//Place your alarm trigger logic here. 
IF io_mapping.cct_3342_b.scaled_value < opc.popa_0082_cct_3342_b_low_setpoint THEN
    cct_3342_b_low.trigger := TRUE;
    ELSE
        cct_3342_b_low.trigger := FALSE;
END_IF
	
//cct_3342-----------------------------------------------------------------------------------------------------
//Instantiate the alarm block, and map the inputs from the OPC GVL
cct_3342_b_high();
cct_3342_b_high.alm_ack:=opc.popa_0082_alarm_ack;
cct_3342_b_high.reset:=opc.popa_0082_alarm_reset;
cct_3342_b_high.priority:=opc.popa_0082_cct_3342_b_high_priority;
cct_3342_b_high.delay_setpoint:=opc.popa_0082_cct_3342_b_high_setpoint;
cct_3342_b_high.enable:=opc.popa_0082_cct_3342_b_high_enable;

//Timer delay elapsed
cct_3342_b_high.delay_ton_et;

//Place your alarm trigger logic here. 
IF io_mapping.cct_3342_b.scaled_value > opc.popa_0082_cct_3342_b_high_setpoint THEN
    cct_3342_b_high.trigger := TRUE;
    ELSE
        cct_3342_b_high.trigger := FALSE;
END_IF
	
//cct_3342-----------------------------------------------------------------------------------------------------
//Instantiate the alarm block, and map the inputs from the OPC GVL
cct_3342_b_high_high();
cct_3342_b_high_high.alm_ack:=opc.popa_0082_alarm_ack;
cct_3342_b_high_high.reset:=opc.popa_0082_alarm_reset;
cct_3342_b_high_high.priority:=opc.popa_0082_cct_3342_b_high_high_priority;
cct_3342_b_high_high.delay_setpoint:=opc.popa_0082_cct_3342_b_high_high_setpoint;
cct_3342_b_high_high.enable:=opc.popa_0082_cct_3342_b_high_high_enable;

//Timer delay elapsed
cct_3342_b_high_high.delay_ton_et;

//Place your alarm trigger logic here. 
IF io_mapping.cct_3342_b.scaled_value >= opc.popa_0082_cct_3342_b_high_high_setpoint THEN
    cct_3342_b_high_high.trigger := TRUE;
    ELSE
        cct_3342_b_high_high.trigger := FALSE;
END_IF

(*
//cct_3413-----------------------------------------------------------------------------------------------------
//Instantiate the alarm block, and map the inputs from the OPC GVL
cct_3413_b_low_low();
cct_3413_b_low_low.alm_ack:=opc.popa_0082_alarm_ack;
cct_3413_b_low_low.reset:=opc.popa_0082_alarm_reset;
cct_3413_b_low_low.priority:=opc.popa_0092_cct_3413_b_low_low_priority;
cct_3413_b_low_low.delay_setpoint:=opc.popa_0092_cct_3413_b_low_low_setpoint;
cct_3413_b_low_low.enable:=opc.popa_0092_cct_3413_b_low_low_enable;

//Timer delay elapsed
cct_3413_b_low_low.delay_ton_et;

//Place your alarm trigger logic here. 
IF io_mapping.cct_3413_b.scaled_value <= opc.popa_0092_cct_3413_b_low_low_setpoint THEN
    cct_3413_b_low_low.trigger := TRUE;
    ELSE
        cct_3413_b_low_low.trigger := FALSE;
END_IF
	
//cct_3413-----------------------------------------------------------------------------------------------------
//Instantiate the alarm block, and map the inputs from the OPC GVL
cct_3413_b_low();
cct_3413_b_low.alm_ack:=opc.popa_0082_alarm_ack;
cct_3413_b_low.reset:=opc.popa_0082_alarm_reset;
cct_3413_b_low.priority:=opc.popa_0092_cct_3413_b_low_priority;
cct_3413_b_low.delay_setpoint:=opc.popa_0092_cct_3413_b_low_setpoint;
cct_3413_b_low.enable:=opc.popa_0092_cct_3413_b_low_enable;

//Timer delay elapsed
cct_3413_b_low.delay_ton_et;

//Place your alarm trigger logic here. 
IF io_mapping.cct_3413_b.scaled_value < opc.popa_0092_cct_3413_b_low_setpoint THEN
    cct_3413_b_low.trigger := TRUE;
    ELSE
        cct_3413_b_low.trigger := FALSE;
END_IF
	
//cct_3413-----------------------------------------------------------------------------------------------------
//Instantiate the alarm block, and map the inputs from the OPC GVL
cct_3413_b_high();
cct_3413_b_high.alm_ack:=opc.popa_0082_alarm_ack;
cct_3413_b_high.reset:=opc.popa_0082_alarm_reset;
cct_3413_b_high.priority:=opc.popa_0092_cct_3413_b_high_priority;
cct_3413_b_high.delay_setpoint:=opc.popa_0092_cct_3413_b_high_setpoint;
cct_3413_b_high.enable:=opc.popa_0092_cct_3413_b_high_enable;

//Timer delay elapsed
cct_3413_b_high.delay_ton_et;

//Place your alarm trigger logic here. 
IF io_mapping.cct_3413_b.scaled_value > opc.popa_0092_cct_3413_b_high_setpoint THEN
    cct_3413_b_high.trigger := TRUE;
    ELSE
        cct_3413_b_high.trigger := FALSE;
END_IF
	
//cct_3413-----------------------------------------------------------------------------------------------------
//Instantiate the alarm block, and map the inputs from the OPC GVL
cct_3413_b_high_high();
cct_3413_b_high_high.alm_ack:=opc.popa_0082_alarm_ack;
cct_3413_b_high_high.reset:=opc.popa_0082_alarm_reset;
cct_3413_b_high_high.priority:=opc.popa_0092_cct_3413_b_high_high_priority;
cct_3413_b_high_high.delay_setpoint:=opc.popa_0092_cct_3413_b_high_high_setpoint;
cct_3413_b_high_high.enable:=opc.popa_0092_cct_3413_b_high_high_enable;

//Timer delay elapsed
cct_3413_b_high_high.delay_ton_et;

//Place your alarm trigger logic here. 
IF io_mapping.cct_3413_b.scaled_value >= opc.popa_0092_cct_3413_b_high_high_setpoint THEN
    cct_3413_b_high_high.trigger := TRUE;
    ELSE
        cct_3413_b_high_high.trigger := FALSE;
END_IF

*)

//ft_3122-----------------------------------------------------------------------------------------------------
//Instantiate the alarm block, and map the inputs from the OPC GVL
ft_3122_b_low_low();
ft_3122_b_low_low.alm_ack:=opc.popa_0082_alarm_ack;
ft_3122_b_low_low.reset:=opc.popa_0082_alarm_reset;
ft_3122_b_low_low.priority:=opc.popa_0082_ft_3122_b_low_low_priority;
ft_3122_b_low_low.delay_setpoint:=opc.popa_0082_ft_3122_b_low_low_setpoint;
ft_3122_b_low_low.enable:=opc.popa_0082_ft_3122_b_low_low_enable;

//Timer delay elapsed
ft_3122_b_low_low.delay_ton_et;

//Place your alarm trigger logic here. 
IF io_mapping.ft_3122_b.scaled_value <= opc.popa_0082_ft_3122_b_low_low_setpoint THEN
    ft_3122_b_low_low.trigger := TRUE;
    ELSE
        ft_3122_b_low_low.trigger := FALSE;
END_IF
	
//ft_3122-----------------------------------------------------------------------------------------------------
//Instantiate the alarm block, and map the inputs from the OPC GVL
ft_3122_b_low();
ft_3122_b_low.alm_ack:=opc.popa_0082_alarm_ack;
ft_3122_b_low.reset:=opc.popa_0082_alarm_reset;
ft_3122_b_low.priority:=opc.popa_0082_ft_3122_b_low_priority;
ft_3122_b_low.delay_setpoint:=opc.popa_0082_ft_3122_b_low_setpoint;
ft_3122_b_low.enable:=opc.popa_0082_ft_3122_b_low_enable;

//Timer delay elapsed
ft_3122_b_low.delay_ton_et;

//Place your alarm trigger logic here. 
IF io_mapping.ft_3122_b.scaled_value < opc.popa_0082_ft_3122_b_low_setpoint THEN
    ft_3122_b_low.trigger := TRUE;
    ELSE
        ft_3122_b_low.trigger := FALSE;
END_IF
	
//ft_3122-----------------------------------------------------------------------------------------------------
//Instantiate the alarm block, and map the inputs from the OPC GVL
ft_3122_b_high();
ft_3122_b_high.alm_ack:=opc.popa_0082_alarm_ack;
ft_3122_b_high.reset:=opc.popa_0082_alarm_reset;
ft_3122_b_high.priority:=opc.popa_0082_ft_3122_b_high_priority;
ft_3122_b_high.delay_setpoint:=opc.popa_0082_ft_3122_b_high_setpoint;
ft_3122_b_high.enable:=opc.popa_0082_ft_3122_b_high_enable;

//Timer delay elapsed
ft_3122_b_high.delay_ton_et;

//Place your alarm trigger logic here. 
IF io_mapping.ft_3122_b.scaled_value > opc.popa_0082_ft_3122_b_high_setpoint THEN
    ft_3122_b_high.trigger := TRUE;
    ELSE
        ft_3122_b_high.trigger := FALSE;
END_IF
	
//ft_3122-----------------------------------------------------------------------------------------------------
//Instantiate the alarm block, and map the inputs from the OPC GVL
ft_3122_b_high_high();
ft_3122_b_high_high.alm_ack:=opc.popa_0082_alarm_ack;
ft_3122_b_high_high.reset:=opc.popa_0082_alarm_reset;
ft_3122_b_high_high.priority:=opc.popa_0082_ft_3122_b_high_high_priority;
ft_3122_b_high_high.delay_setpoint:=opc.popa_0082_ft_3122_b_high_high_setpoint;
ft_3122_b_high_high.enable:=opc.popa_0082_ft_3122_b_high_high_enable;

//Timer delay elapsed
ft_3122_b_high_high.delay_ton_et;

//Place your alarm trigger logic here. 
IF io_mapping.ft_3122_b.scaled_value >= opc.popa_0082_ft_3122_b_high_high_setpoint THEN
    ft_3122_b_high_high.trigger := TRUE;
    ELSE
        ft_3122_b_high_high.trigger := FALSE;
END_IF


//ft_3222-----------------------------------------------------------------------------------------------------
//Instantiate the alarm block, and map the inputs from the OPC GVL
ft_3222_b_low_low();
ft_3222_b_low_low.alm_ack:=opc.popa_0082_alarm_ack;
ft_3222_b_low_low.reset:=opc.popa_0082_alarm_reset;
ft_3222_b_low_low.priority:=opc.popa_0082_ft_3222_b_low_low_priority;
ft_3222_b_low_low.delay_setpoint:=opc.popa_0082_ft_3222_b_low_low_setpoint;
ft_3222_b_low_low.enable:=opc.popa_0082_ft_3222_b_low_low_enable;

//Timer delay elapsed
ft_3222_b_low_low.delay_ton_et;

//Place your alarm trigger logic here. 
IF io_mapping.ft_3222_b.scaled_value <= opc.popa_0082_ft_3222_b_low_low_setpoint THEN
    ft_3222_b_low_low.trigger := TRUE;
    ELSE
        ft_3222_b_low_low.trigger := FALSE;
END_IF
	
//ft_3222-----------------------------------------------------------------------------------------------------
//Instantiate the alarm block, and map the inputs from the OPC GVL
ft_3222_b_low();
ft_3222_b_low.alm_ack:=opc.popa_0082_alarm_ack;
ft_3222_b_low.reset:=opc.popa_0082_alarm_reset;
ft_3222_b_low.priority:=opc.popa_0082_ft_3222_b_low_priority;
ft_3222_b_low.delay_setpoint:=opc.popa_0082_ft_3222_b_low_setpoint;
ft_3222_b_low.enable:=opc.popa_0082_ft_3222_b_low_enable;

//Timer delay elapsed
ft_3222_b_low.delay_ton_et;

//Place your alarm trigger logic here. 
IF io_mapping.ft_3222_b.scaled_value < opc.popa_0082_ft_3222_b_low_setpoint THEN
    ft_3222_b_low.trigger := TRUE;
    ELSE
        ft_3222_b_low.trigger := FALSE;
END_IF
	
//ft_3222-----------------------------------------------------------------------------------------------------
//Instantiate the alarm block, and map the inputs from the OPC GVL
ft_3222_b_high();
ft_3222_b_high.alm_ack:=opc.popa_0082_alarm_ack;
ft_3222_b_high.reset:=opc.popa_0082_alarm_reset;
ft_3222_b_high.priority:=opc.popa_0082_ft_3222_b_high_priority;
ft_3222_b_high.delay_setpoint:=opc.popa_0082_ft_3222_b_high_setpoint;
ft_3222_b_high.enable:=opc.popa_0082_ft_3222_b_high_enable;

//Timer delay elapsed
ft_3222_b_high.delay_ton_et;

//Place your alarm trigger logic here. 
IF io_mapping.ft_3222_b.scaled_value > opc.popa_0082_ft_3222_b_high_setpoint THEN
    ft_3222_b_high.trigger := TRUE;
    ELSE
        ft_3222_b_high.trigger := FALSE;
END_IF
	
//ft_3222-----------------------------------------------------------------------------------------------------
//Instantiate the alarm block, and map the inputs from the OPC GVL
ft_3222_b_high_high();
ft_3222_b_high_high.alm_ack:=opc.popa_0082_alarm_ack;
ft_3222_b_high_high.reset:=opc.popa_0082_alarm_reset;
ft_3222_b_high_high.priority:=opc.popa_0082_ft_3222_b_high_high_priority;
ft_3222_b_high_high.delay_setpoint:=opc.popa_0082_ft_3222_b_high_high_setpoint;
ft_3222_b_high_high.enable:=opc.popa_0082_ft_3222_b_high_high_enable;

//Timer delay elapsed
ft_3222_b_high_high.delay_ton_et;

//Place your alarm trigger logic here. 
IF io_mapping.ft_3222_b.scaled_value >= opc.popa_0082_ft_3222_b_high_high_setpoint THEN
    ft_3222_b_high_high.trigger := TRUE;
    ELSE
        ft_3222_b_high_high.trigger := FALSE;
END_IF


//ft_3322-----------------------------------------------------------------------------------------------------
//Instantiate the alarm block, and map the inputs from the OPC GVL
ft_3322_b_low_low();
ft_3322_b_low_low.alm_ack:=opc.popa_0082_alarm_ack;
ft_3322_b_low_low.reset:=opc.popa_0082_alarm_reset;
ft_3322_b_low_low.priority:=opc.popa_0082_ft_3322_b_low_low_priority;
ft_3322_b_low_low.delay_setpoint:=opc.popa_0082_ft_3322_b_low_low_setpoint;
ft_3322_b_low_low.enable:=opc.popa_0082_ft_3322_b_low_low_enable;

//Timer delay elapsed
ft_3322_b_low_low.delay_ton_et;

//Place your alarm trigger logic here. 
IF io_mapping.ft_3322_b.scaled_value <= opc.popa_0082_ft_3322_b_low_low_setpoint THEN
    ft_3322_b_low_low.trigger := TRUE;
    ELSE
        ft_3322_b_low_low.trigger := FALSE;
END_IF
	
//ft_3322-----------------------------------------------------------------------------------------------------
//Instantiate the alarm block, and map the inputs from the OPC GVL
ft_3322_b_low();
ft_3322_b_low.alm_ack:=opc.popa_0082_alarm_ack;
ft_3322_b_low.reset:=opc.popa_0082_alarm_reset;
ft_3322_b_low.priority:=opc.popa_0082_ft_3322_b_low_priority;
ft_3322_b_low.delay_setpoint:=opc.popa_0082_ft_3322_b_low_setpoint;
ft_3322_b_low.enable:=opc.popa_0082_ft_3322_b_low_enable;

//Timer delay elapsed
ft_3322_b_low.delay_ton_et;

//Place your alarm trigger logic here. 
IF io_mapping.ft_3322_b.scaled_value < opc.popa_0082_ft_3322_b_low_setpoint THEN
    ft_3322_b_low.trigger := TRUE;
    ELSE
        ft_3322_b_low.trigger := FALSE;
END_IF
	
//ft_3322-----------------------------------------------------------------------------------------------------
//Instantiate the alarm block, and map the inputs from the OPC GVL
ft_3322_b_high();
ft_3322_b_high.alm_ack:=opc.popa_0082_alarm_ack;
ft_3322_b_high.reset:=opc.popa_0082_alarm_reset;
ft_3322_b_high.priority:=opc.popa_0082_ft_3322_b_high_priority;
ft_3322_b_high.delay_setpoint:=opc.popa_0082_ft_3322_b_high_setpoint;
ft_3322_b_high.enable:=opc.popa_0082_ft_3322_b_high_enable;

//Timer delay elapsed
ft_3322_b_high.delay_ton_et;

//Place your alarm trigger logic here. 
IF io_mapping.ft_3322_b.scaled_value > opc.popa_0082_ft_3322_b_high_setpoint THEN
    ft_3322_b_high.trigger := TRUE;
    ELSE
        ft_3322_b_high.trigger := FALSE;
END_IF
	
//ft_3322-----------------------------------------------------------------------------------------------------
//Instantiate the alarm block, and map the inputs from the OPC GVL
ft_3322_b_high_high();
ft_3322_b_high_high.alm_ack:=opc.popa_0082_alarm_ack;
ft_3322_b_high_high.reset:=opc.popa_0082_alarm_reset;
ft_3322_b_high_high.priority:=opc.popa_0082_ft_3322_b_high_high_priority;
ft_3322_b_high_high.delay_setpoint:=opc.popa_0082_ft_3322_b_high_high_setpoint;
ft_3322_b_high_high.enable:=opc.popa_0082_ft_3322_b_high_high_enable;

//Timer delay elapsed
ft_3322_b_high_high.delay_ton_et;

//Place your alarm trigger logic here. 
IF io_mapping.ft_3322_b.scaled_value >= opc.popa_0082_ft_3322_b_high_high_setpoint THEN
    ft_3322_b_high_high.trigger := TRUE;
    ELSE
        ft_3322_b_high_high.trigger := FALSE;
END_IF


//lt_3102-----------------------------------------------------------------------------------------------------
//Instantiate the alarm block, and map the inputs from the OPC GVL
lt_3102_b_low_low();
lt_3102_b_low_low.alm_ack:=opc.popa_0082_alarm_ack;
lt_3102_b_low_low.reset:=opc.popa_0082_alarm_reset;
lt_3102_b_low_low.priority:=opc.popa_0082_lt_3102_b_low_low_priority;
lt_3102_b_low_low.delay_setpoint:=opc.popa_0082_lt_3102_b_low_low_setpoint;
lt_3102_b_low_low.enable:=opc.popa_0082_lt_3102_b_low_low_enable;

//Timer delay elapsed
lt_3102_b_low_low.delay_ton_et;

//Place your alarm trigger logic here. 
IF io_mapping.lt_3102_b.scaled_value <= opc.popa_0082_lt_3102_b_low_low_setpoint THEN
    lt_3102_b_low_low.trigger := TRUE;
    ELSE
        lt_3102_b_low_low.trigger := FALSE;
END_IF
	
//lt_3102-----------------------------------------------------------------------------------------------------
//Instantiate the alarm block, and map the inputs from the OPC GVL
lt_3102_b_low();
lt_3102_b_low.alm_ack:=opc.popa_0082_alarm_ack;
lt_3102_b_low.reset:=opc.popa_0082_alarm_reset;
lt_3102_b_low.priority:=opc.popa_0082_lt_3102_b_low_priority;
lt_3102_b_low.delay_setpoint:=opc.popa_0082_lt_3102_b_low_setpoint;
lt_3102_b_low.enable:=opc.popa_0082_lt_3102_b_low_enable;

//Timer delay elapsed
lt_3102_b_low.delay_ton_et;

//Place your alarm trigger logic here. 
IF io_mapping.lt_3102_b.scaled_value < opc.popa_0082_lt_3102_b_low_setpoint THEN
    lt_3102_b_low.trigger := TRUE;
    ELSE
        lt_3102_b_low.trigger := FALSE;
END_IF
	
//lt_3102-----------------------------------------------------------------------------------------------------
//Instantiate the alarm block, and map the inputs from the OPC GVL
lt_3102_b_high();
lt_3102_b_high.alm_ack:=opc.popa_0082_alarm_ack;
lt_3102_b_high.reset:=opc.popa_0082_alarm_reset;
lt_3102_b_high.priority:=opc.popa_0082_lt_3102_b_high_priority;
lt_3102_b_high.delay_setpoint:=opc.popa_0082_lt_3102_b_high_setpoint;
lt_3102_b_high.enable:=opc.popa_0082_lt_3102_b_high_enable;

//Timer delay elapsed
lt_3102_b_high.delay_ton_et;

//Place your alarm trigger logic here. 
IF io_mapping.lt_3102_b.scaled_value > opc.popa_0082_lt_3102_b_high_setpoint THEN
    lt_3102_b_high.trigger := TRUE;
    ELSE
        lt_3102_b_high.trigger := FALSE;
END_IF
	
//lt_3102-----------------------------------------------------------------------------------------------------
//Instantiate the alarm block, and map the inputs from the OPC GVL
lt_3102_b_high_high();
lt_3102_b_high_high.alm_ack:=opc.popa_0082_alarm_ack;
lt_3102_b_high_high.reset:=opc.popa_0082_alarm_reset;
lt_3102_b_high_high.priority:=opc.popa_0082_lt_3102_b_high_high_priority;
lt_3102_b_high_high.delay_setpoint:=opc.popa_0082_lt_3102_b_high_high_setpoint;
lt_3102_b_high_high.enable:=opc.popa_0082_lt_3102_b_high_high_enable;

//Timer delay elapsed
lt_3102_b_high_high.delay_ton_et;

//Place your alarm trigger logic here. 
IF io_mapping.lt_3102_b.scaled_value >= opc.popa_0082_lt_3102_b_high_high_setpoint THEN
    lt_3102_b_high_high.trigger := TRUE;
    ELSE
        lt_3102_b_high_high.trigger := FALSE;
END_IF


//lt_3202-----------------------------------------------------------------------------------------------------
//Instantiate the alarm block, and map the inputs from the OPC GVL
lt_3202_b_low_low();
lt_3202_b_low_low.alm_ack:=opc.popa_0082_alarm_ack;
lt_3202_b_low_low.reset:=opc.popa_0082_alarm_reset;
lt_3202_b_low_low.priority:=opc.popa_0082_lt_3202_b_low_low_priority;
lt_3202_b_low_low.delay_setpoint:=opc.popa_0082_lt_3202_b_low_low_setpoint;
lt_3202_b_low_low.enable:=opc.popa_0082_lt_3202_b_low_low_enable;

//Timer delay elapsed
lt_3202_b_low_low.delay_ton_et;

//Place your alarm trigger logic here. 
IF io_mapping.lt_3202_b.scaled_value <= opc.popa_0082_lt_3202_b_low_low_setpoint THEN
    lt_3202_b_low_low.trigger := TRUE;
    ELSE
        lt_3202_b_low_low.trigger := FALSE;
END_IF
	
//lt_3202-----------------------------------------------------------------------------------------------------
//Instantiate the alarm block, and map the inputs from the OPC GVL
lt_3202_b_low();
lt_3202_b_low.alm_ack:=opc.popa_0082_alarm_ack;
lt_3202_b_low.reset:=opc.popa_0082_alarm_reset;
lt_3202_b_low.priority:=opc.popa_0082_lt_3202_b_low_priority;
lt_3202_b_low.delay_setpoint:=opc.popa_0082_lt_3202_b_low_setpoint;
lt_3202_b_low.enable:=opc.popa_0082_lt_3202_b_low_enable;

//Timer delay elapsed
lt_3202_b_low.delay_ton_et;

//Place your alarm trigger logic here. 
IF io_mapping.lt_3202_b.scaled_value < opc.popa_0082_lt_3202_b_low_setpoint THEN
    lt_3202_b_low.trigger := TRUE;
    ELSE
        lt_3202_b_low.trigger := FALSE;
END_IF
	
//lt_3202-----------------------------------------------------------------------------------------------------
//Instantiate the alarm block, and map the inputs from the OPC GVL
lt_3202_b_high();
lt_3202_b_high.alm_ack:=opc.popa_0082_alarm_ack;
lt_3202_b_high.reset:=opc.popa_0082_alarm_reset;
lt_3202_b_high.priority:=opc.popa_0082_lt_3202_b_high_priority;
lt_3202_b_high.delay_setpoint:=opc.popa_0082_lt_3202_b_high_setpoint;
lt_3202_b_high.enable:=opc.popa_0082_lt_3202_b_high_enable;

//Timer delay elapsed
lt_3202_b_high.delay_ton_et;

//Place your alarm trigger logic here. 
IF io_mapping.lt_3202_b.scaled_value > opc.popa_0082_lt_3202_b_high_setpoint THEN
    lt_3202_b_high.trigger := TRUE;
    ELSE
        lt_3202_b_high.trigger := FALSE;
END_IF
	
//lt_3202-----------------------------------------------------------------------------------------------------
//Instantiate the alarm block, and map the inputs from the OPC GVL
lt_3202_b_high_high();
lt_3202_b_high_high.alm_ack:=opc.popa_0082_alarm_ack;
lt_3202_b_high_high.reset:=opc.popa_0082_alarm_reset;
lt_3202_b_high_high.priority:=opc.popa_0082_lt_3202_b_high_high_priority;
lt_3202_b_high_high.delay_setpoint:=opc.popa_0082_lt_3202_b_high_high_setpoint;
lt_3202_b_high_high.enable:=opc.popa_0082_lt_3202_b_high_high_enable;

//Timer delay elapsed
lt_3202_b_high_high.delay_ton_et;

//Place your alarm trigger logic here. 
IF io_mapping.lt_3202_b.scaled_value >= opc.popa_0082_lt_3202_b_high_high_setpoint THEN
    lt_3202_b_high_high.trigger := TRUE;
    ELSE
        lt_3202_b_high_high.trigger := FALSE;
END_IF


//lt_3302-----------------------------------------------------------------------------------------------------
//Instantiate the alarm block, and map the inputs from the OPC GVL
lt_3302_b_low_low();
lt_3302_b_low_low.alm_ack:=opc.popa_0082_alarm_ack;
lt_3302_b_low_low.reset:=opc.popa_0082_alarm_reset;
lt_3302_b_low_low.priority:=opc.popa_0082_lt_3302_b_low_low_priority;
lt_3302_b_low_low.delay_setpoint:=opc.popa_0082_lt_3302_b_low_low_setpoint;
lt_3302_b_low_low.enable:=opc.popa_0082_lt_3302_b_low_low_enable;

//Timer delay elapsed
lt_3302_b_low_low.delay_ton_et;

//Place your alarm trigger logic here. 
IF io_mapping.lt_3302_b.scaled_value <= opc.popa_0082_lt_3302_b_low_low_setpoint THEN
    lt_3302_b_low_low.trigger := TRUE;
    ELSE
        lt_3302_b_low_low.trigger := FALSE;
END_IF
	
//lt_3302-----------------------------------------------------------------------------------------------------
//Instantiate the alarm block, and map the inputs from the OPC GVL
lt_3302_b_low();
lt_3302_b_low.alm_ack:=opc.popa_0082_alarm_ack;
lt_3302_b_low.reset:=opc.popa_0082_alarm_reset;
lt_3302_b_low.priority:=opc.popa_0082_lt_3302_b_low_priority;
lt_3302_b_low.delay_setpoint:=opc.popa_0082_lt_3302_b_low_setpoint;
lt_3302_b_low.enable:=opc.popa_0082_lt_3302_b_low_enable;

//Timer delay elapsed
lt_3302_b_low.delay_ton_et;

//Place your alarm trigger logic here. 
IF io_mapping.lt_3302_b.scaled_value < opc.popa_0082_lt_3302_b_low_setpoint THEN
    lt_3302_b_low.trigger := TRUE;
    ELSE
        lt_3302_b_low.trigger := FALSE;
END_IF
	
//lt_3302-----------------------------------------------------------------------------------------------------
//Instantiate the alarm block, and map the inputs from the OPC GVL
lt_3302_b_high();
lt_3302_b_high.alm_ack:=opc.popa_0082_alarm_ack;
lt_3302_b_high.reset:=opc.popa_0082_alarm_reset;
lt_3302_b_high.priority:=opc.popa_0082_lt_3302_b_high_priority;
lt_3302_b_high.delay_setpoint:=opc.popa_0082_lt_3302_b_high_setpoint;
lt_3302_b_high.enable:=opc.popa_0082_lt_3302_b_high_enable;

//Timer delay elapsed
lt_3302_b_high.delay_ton_et;

//Place your alarm trigger logic here. 
IF io_mapping.lt_3302_b.scaled_value > opc.popa_0082_lt_3302_b_high_setpoint THEN
    lt_3302_b_high.trigger := TRUE;
    ELSE
        lt_3302_b_high.trigger := FALSE;
END_IF
	
//lt_3302-----------------------------------------------------------------------------------------------------
//Instantiate the alarm block, and map the inputs from the OPC GVL
lt_3302_b_high_high();
lt_3302_b_high_high.alm_ack:=opc.popa_0082_alarm_ack;
lt_3302_b_high_high.reset:=opc.popa_0082_alarm_reset;
lt_3302_b_high_high.priority:=opc.popa_0082_lt_3302_b_high_high_priority;
lt_3302_b_high_high.delay_setpoint:=opc.popa_0082_lt_3302_b_high_high_setpoint;
lt_3302_b_high_high.enable:=opc.popa_0082_lt_3302_b_high_high_enable;

//Timer delay elapsed
lt_3302_b_high_high.delay_ton_et;

//Place your alarm trigger logic here. 
IF io_mapping.lt_3302_b.scaled_value >= opc.popa_0082_lt_3302_b_high_high_setpoint THEN
    lt_3302_b_high_high.trigger := TRUE;
    ELSE
        lt_3302_b_high_high.trigger := FALSE;
END_IF


//lt_3153-----------------------------------------------------------------------------------------------------
//Instantiate the alarm block, and map the inputs from the OPC GVL
lt_3153_b_low_low();
lt_3153_b_low_low.alm_ack:=opc.popa_0082_alarm_ack;
lt_3153_b_low_low.reset:=opc.popa_0082_alarm_reset;
lt_3153_b_low_low.priority:=opc.popa_0082_lt_3153_b_low_low_priority;
lt_3153_b_low_low.delay_setpoint:=opc.popa_0082_lt_3153_b_low_low_setpoint;
lt_3153_b_low_low.enable:=opc.popa_0082_lt_3153_b_low_low_enable;

//Timer delay elapsed
lt_3153_b_low_low.delay_ton_et;

//Place your alarm trigger logic here. 
IF io_mapping.lt_3153_b.scaled_value <= opc.popa_0082_lt_3153_b_low_low_setpoint THEN
    lt_3153_b_low_low.trigger := TRUE;
    ELSE
        lt_3153_b_low_low.trigger := FALSE;
END_IF
	
//lt_3153-----------------------------------------------------------------------------------------------------
//Instantiate the alarm block, and map the inputs from the OPC GVL
lt_3153_b_low();
lt_3153_b_low.alm_ack:=opc.popa_0082_alarm_ack;
lt_3153_b_low.reset:=opc.popa_0082_alarm_reset;
lt_3153_b_low.priority:=opc.popa_0082_lt_3153_b_low_priority;
lt_3153_b_low.delay_setpoint:=opc.popa_0082_lt_3153_b_low_setpoint;
lt_3153_b_low.enable:=opc.popa_0082_lt_3153_b_low_enable;

//Timer delay elapsed
lt_3153_b_low.delay_ton_et;

//Place your alarm trigger logic here. 
IF io_mapping.lt_3153_b.scaled_value < opc.popa_0082_lt_3153_b_low_setpoint THEN
    lt_3153_b_low.trigger := TRUE;
    ELSE
        lt_3153_b_low.trigger := FALSE;
END_IF
	
//lt_3153-----------------------------------------------------------------------------------------------------
//Instantiate the alarm block, and map the inputs from the OPC GVL
lt_3153_b_high();
lt_3153_b_high.alm_ack:=opc.popa_0082_alarm_ack;
lt_3153_b_high.reset:=opc.popa_0082_alarm_reset;
lt_3153_b_high.priority:=opc.popa_0082_lt_3153_b_high_priority;
lt_3153_b_high.delay_setpoint:=opc.popa_0082_lt_3153_b_high_setpoint;
lt_3153_b_high.enable:=opc.popa_0082_lt_3153_b_high_enable;

//Timer delay elapsed
lt_3153_b_high.delay_ton_et;

//Place your alarm trigger logic here. 
IF io_mapping.lt_3153_b.scaled_value > opc.popa_0082_lt_3153_b_high_setpoint THEN
    lt_3153_b_high.trigger := TRUE;
    ELSE
        lt_3153_b_high.trigger := FALSE;
END_IF
	
//lt_3153-----------------------------------------------------------------------------------------------------
//Instantiate the alarm block, and map the inputs from the OPC GVL
lt_3153_b_high_high();
lt_3153_b_high_high.alm_ack:=opc.popa_0082_alarm_ack;
lt_3153_b_high_high.reset:=opc.popa_0082_alarm_reset;
lt_3153_b_high_high.priority:=opc.popa_0082_lt_3153_b_high_high_priority;
lt_3153_b_high_high.delay_setpoint:=opc.popa_0082_lt_3153_b_high_high_setpoint;
lt_3153_b_high_high.enable:=opc.popa_0082_lt_3153_b_high_high_enable;

//Timer delay elapsed
lt_3153_b_high_high.delay_ton_et;

//Place your alarm trigger logic here. 
IF io_mapping.lt_3153_b.scaled_value >= opc.popa_0082_lt_3153_b_high_high_setpoint THEN
    lt_3153_b_high_high.trigger := TRUE;
    ELSE
        lt_3153_b_high_high.trigger := FALSE;
END_IF


//lt_3253-----------------------------------------------------------------------------------------------------
//Instantiate the alarm block, and map the inputs from the OPC GVL
lt_3253_b_low_low();
lt_3253_b_low_low.alm_ack:=opc.popa_0082_alarm_ack;
lt_3253_b_low_low.reset:=opc.popa_0082_alarm_reset;
lt_3253_b_low_low.priority:=opc.popa_0082_lt_3253_b_low_low_priority;
lt_3253_b_low_low.delay_setpoint:=opc.popa_0082_lt_3253_b_low_low_setpoint;
lt_3253_b_low_low.enable:=opc.popa_0082_lt_3253_b_low_low_enable;

//Timer delay elapsed
lt_3253_b_low_low.delay_ton_et;

//Place your alarm trigger logic here. 
IF io_mapping.lt_3253_b.scaled_value <= opc.popa_0082_lt_3253_b_low_low_setpoint THEN
    lt_3253_b_low_low.trigger := TRUE;
    ELSE
        lt_3253_b_low_low.trigger := FALSE;
END_IF
	
//lt_3253-----------------------------------------------------------------------------------------------------
//Instantiate the alarm block, and map the inputs from the OPC GVL
lt_3253_b_low();
lt_3253_b_low.alm_ack:=opc.popa_0082_alarm_ack;
lt_3253_b_low.reset:=opc.popa_0082_alarm_reset;
lt_3253_b_low.priority:=opc.popa_0082_lt_3253_b_low_priority;
lt_3253_b_low.delay_setpoint:=opc.popa_0082_lt_3253_b_low_setpoint;
lt_3253_b_low.enable:=opc.popa_0082_lt_3253_b_low_enable;

//Timer delay elapsed
lt_3253_b_low.delay_ton_et;

//Place your alarm trigger logic here. 
IF io_mapping.lt_3253_b.scaled_value < opc.popa_0082_lt_3253_b_low_setpoint THEN
    lt_3253_b_low.trigger := TRUE;
    ELSE
        lt_3253_b_low.trigger := FALSE;
END_IF
	
//lt_3253-----------------------------------------------------------------------------------------------------
//Instantiate the alarm block, and map the inputs from the OPC GVL
lt_3253_b_high();
lt_3253_b_high.alm_ack:=opc.popa_0082_alarm_ack;
lt_3253_b_high.reset:=opc.popa_0082_alarm_reset;
lt_3253_b_high.priority:=opc.popa_0082_lt_3253_b_high_priority;
lt_3253_b_high.delay_setpoint:=opc.popa_0082_lt_3253_b_high_setpoint;
lt_3253_b_high.enable:=opc.popa_0082_lt_3253_b_high_enable;

//Timer delay elapsed
lt_3253_b_high.delay_ton_et;

//Place your alarm trigger logic here. 
IF io_mapping.lt_3253_b.scaled_value > opc.popa_0082_lt_3253_b_high_setpoint THEN
    lt_3253_b_high.trigger := TRUE;
    ELSE
        lt_3253_b_high.trigger := FALSE;
END_IF
	
//lt_3253-----------------------------------------------------------------------------------------------------
//Instantiate the alarm block, and map the inputs from the OPC GVL
lt_3253_b_high_high();
lt_3253_b_high_high.alm_ack:=opc.popa_0082_alarm_ack;
lt_3253_b_high_high.reset:=opc.popa_0082_alarm_reset;
lt_3253_b_high_high.priority:=opc.popa_0082_lt_3253_b_high_high_priority;
lt_3253_b_high_high.delay_setpoint:=opc.popa_0082_lt_3253_b_high_high_setpoint;
lt_3253_b_high_high.enable:=opc.popa_0082_lt_3253_b_high_high_enable;

//Timer delay elapsed
lt_3253_b_high_high.delay_ton_et;

//Place your alarm trigger logic here. 
IF io_mapping.lt_3253_b.scaled_value >= opc.popa_0082_lt_3253_b_high_high_setpoint THEN
    lt_3253_b_high_high.trigger := TRUE;
    ELSE
        lt_3253_b_high_high.trigger := FALSE;
END_IF


//lt_3353-----------------------------------------------------------------------------------------------------
//Instantiate the alarm block, and map the inputs from the OPC GVL
lt_3353_b_low_low();
lt_3353_b_low_low.alm_ack:=opc.popa_0082_alarm_ack;
lt_3353_b_low_low.reset:=opc.popa_0082_alarm_reset;
lt_3353_b_low_low.priority:=opc.popa_0082_lt_3353_b_low_low_priority;
lt_3353_b_low_low.delay_setpoint:=opc.popa_0082_lt_3353_b_low_low_setpoint;
lt_3353_b_low_low.enable:=opc.popa_0082_lt_3353_b_low_low_enable;

//Timer delay elapsed
lt_3353_b_low_low.delay_ton_et;

//Place your alarm trigger logic here. 
IF io_mapping.lt_3353_b.scaled_value <= opc.popa_0082_lt_3353_b_low_low_setpoint THEN
    lt_3353_b_low_low.trigger := TRUE;
    ELSE
        lt_3353_b_low_low.trigger := FALSE;
END_IF
	
//lt_3353-----------------------------------------------------------------------------------------------------
//Instantiate the alarm block, and map the inputs from the OPC GVL
lt_3353_b_low();
lt_3353_b_low.alm_ack:=opc.popa_0082_alarm_ack;
lt_3353_b_low.reset:=opc.popa_0082_alarm_reset;
lt_3353_b_low.priority:=opc.popa_0082_lt_3353_b_low_priority;
lt_3353_b_low.delay_setpoint:=opc.popa_0082_lt_3353_b_low_setpoint;
lt_3353_b_low.enable:=opc.popa_0082_lt_3353_b_low_enable;

//Timer delay elapsed
lt_3353_b_low.delay_ton_et;

//Place your alarm trigger logic here. 
IF io_mapping.lt_3353_b.scaled_value < opc.popa_0082_lt_3353_b_low_setpoint THEN
    lt_3353_b_low.trigger := TRUE;
    ELSE
        lt_3353_b_low.trigger := FALSE;
END_IF
	
//lt_3353-----------------------------------------------------------------------------------------------------
//Instantiate the alarm block, and map the inputs from the OPC GVL
lt_3353_b_high();
lt_3353_b_high.alm_ack:=opc.popa_0082_alarm_ack;
lt_3353_b_high.reset:=opc.popa_0082_alarm_reset;
lt_3353_b_high.priority:=opc.popa_0082_lt_3353_b_high_priority;
lt_3353_b_high.delay_setpoint:=opc.popa_0082_lt_3353_b_high_setpoint;
lt_3353_b_high.enable:=opc.popa_0082_lt_3353_b_high_enable;

//Timer delay elapsed
lt_3353_b_high.delay_ton_et;

//Place your alarm trigger logic here. 
IF io_mapping.lt_3353_b.scaled_value > opc.popa_0082_lt_3353_b_high_setpoint THEN
    lt_3353_b_high.trigger := TRUE;
    ELSE
        lt_3353_b_high.trigger := FALSE;
END_IF
	
//lt_3353-----------------------------------------------------------------------------------------------------
//Instantiate the alarm block, and map the inputs from the OPC GVL
lt_3353_b_high_high();
lt_3353_b_high_high.alm_ack:=opc.popa_0082_alarm_ack;
lt_3353_b_high_high.reset:=opc.popa_0082_alarm_reset;
lt_3353_b_high_high.priority:=opc.popa_0082_lt_3353_b_high_high_priority;
lt_3353_b_high_high.delay_setpoint:=opc.popa_0082_lt_3353_b_high_high_setpoint;
lt_3353_b_high_high.enable:=opc.popa_0082_lt_3353_b_high_high_enable;

//Timer delay elapsed
lt_3353_b_high_high.delay_ton_et;

//Place your alarm trigger logic here. 
IF io_mapping.lt_3353_b.scaled_value >= opc.popa_0082_lt_3353_b_high_high_setpoint THEN
    lt_3353_b_high_high.trigger := TRUE;
    ELSE
        lt_3353_b_high_high.trigger := FALSE;
END_IF


//lt_3402-----------------------------------------------------------------------------------------------------
//Instantiate the alarm block, and map the inputs from the OPC GVL
lt_3402_b_low_low();
lt_3402_b_low_low.alm_ack:=opc.popa_0082_alarm_ack;
lt_3402_b_low_low.reset:=opc.popa_0082_alarm_reset;
lt_3402_b_low_low.priority:=opc.popa_0092_lt_3402_b_low_low_priority;
lt_3402_b_low_low.delay_setpoint:=opc.popa_0092_lt_3402_b_low_low_setpoint;
lt_3402_b_low_low.enable:=opc.popa_0092_lt_3402_b_low_low_enable;

//Timer delay elapsed
lt_3402_b_low_low.delay_ton_et;

//Place your alarm trigger logic here. 
IF io_mapping.lt_3402_b.scaled_value <= opc.popa_0092_lt_3402_b_low_low_setpoint THEN
    lt_3402_b_low_low.trigger := TRUE;
    ELSE
        lt_3402_b_low_low.trigger := FALSE;
END_IF
	
//lt_3402-----------------------------------------------------------------------------------------------------
//Instantiate the alarm block, and map the inputs from the OPC GVL
lt_3402_b_low();
lt_3402_b_low.alm_ack:=opc.popa_0082_alarm_ack;
lt_3402_b_low.reset:=opc.popa_0082_alarm_reset;
lt_3402_b_low.priority:=opc.popa_0092_lt_3402_b_low_priority;
lt_3402_b_low.delay_setpoint:=opc.popa_0092_lt_3402_b_low_setpoint;
lt_3402_b_low.enable:=opc.popa_0092_lt_3402_b_low_enable;

//Timer delay elapsed
lt_3402_b_low.delay_ton_et;

//Place your alarm trigger logic here. 
IF io_mapping.lt_3402_b.scaled_value < opc.popa_0092_lt_3402_b_low_setpoint THEN
    lt_3402_b_low.trigger := TRUE;
    ELSE
        lt_3402_b_low.trigger := FALSE;
END_IF
	
//lt_3402-----------------------------------------------------------------------------------------------------
//Instantiate the alarm block, and map the inputs from the OPC GVL
lt_3402_b_high();
lt_3402_b_high.alm_ack:=opc.popa_0082_alarm_ack;
lt_3402_b_high.reset:=opc.popa_0082_alarm_reset;
lt_3402_b_high.priority:=opc.popa_0092_lt_3402_b_high_priority;
lt_3402_b_high.delay_setpoint:=opc.popa_0092_lt_3402_b_high_setpoint;
lt_3402_b_high.enable:=opc.popa_0092_lt_3402_b_high_enable;

//Timer delay elapsed
lt_3402_b_high.delay_ton_et;

//Place your alarm trigger logic here. 
IF io_mapping.lt_3402_b.scaled_value > opc.popa_0092_lt_3402_b_high_setpoint THEN
    lt_3402_b_high.trigger := TRUE;
    ELSE
        lt_3402_b_high.trigger := FALSE;
END_IF
	
//lt_3402-----------------------------------------------------------------------------------------------------
//Instantiate the alarm block, and map the inputs from the OPC GVL
lt_3402_b_high_high();
lt_3402_b_high_high.alm_ack:=opc.popa_0082_alarm_ack;
lt_3402_b_high_high.reset:=opc.popa_0082_alarm_reset;
lt_3402_b_high_high.priority:=opc.popa_0092_lt_3402_b_high_high_priority;
lt_3402_b_high_high.delay_setpoint:=opc.popa_0092_lt_3402_b_high_high_setpoint;
lt_3402_b_high_high.enable:=opc.popa_0092_lt_3402_b_high_high_enable;

//Timer delay elapsed
lt_3402_b_high_high.delay_ton_et;

//Place your alarm trigger logic here. 
IF io_mapping.lt_3402_b.scaled_value >= opc.popa_0092_lt_3402_b_high_high_setpoint THEN
    lt_3402_b_high_high.trigger := TRUE;
    ELSE
        lt_3402_b_high_high.trigger := FALSE;
END_IF


//pt_3119-----------------------------------------------------------------------------------------------------
//Instantiate the alarm block, and map the inputs from the OPC GVL
pt_3119_b_low_low();
pt_3119_b_low_low.alm_ack:=opc.popa_0082_alarm_ack;
pt_3119_b_low_low.reset:=opc.popa_0082_alarm_reset;
pt_3119_b_low_low.priority:=opc.popa_0082_pt_3119_b_low_low_priority;
pt_3119_b_low_low.delay_setpoint:=opc.popa_0082_pt_3119_b_low_low_setpoint;
pt_3119_b_low_low.enable:=opc.popa_0082_pt_3119_b_low_low_enable;

//Timer delay elapsed
pt_3119_b_low_low.delay_ton_et;

//Place your alarm trigger logic here. 
IF io_mapping.pt_3119_b.scaled_value <= opc.popa_0082_pt_3119_b_low_low_setpoint THEN
    pt_3119_b_low_low.trigger := TRUE;
    ELSE
        pt_3119_b_low_low.trigger := FALSE;
END_IF
	
//pt_3119-----------------------------------------------------------------------------------------------------
//Instantiate the alarm block, and map the inputs from the OPC GVL
pt_3119_b_low();
pt_3119_b_low.alm_ack:=opc.popa_0082_alarm_ack;
pt_3119_b_low.reset:=opc.popa_0082_alarm_reset;
pt_3119_b_low.priority:=opc.popa_0082_pt_3119_b_low_priority;
pt_3119_b_low.delay_setpoint:=opc.popa_0082_pt_3119_b_low_setpoint;
pt_3119_b_low.enable:=opc.popa_0082_pt_3119_b_low_enable;

//Timer delay elapsed
pt_3119_b_low.delay_ton_et;

//Place your alarm trigger logic here. 
IF io_mapping.pt_3119_b.scaled_value < opc.popa_0082_pt_3119_b_low_setpoint THEN
    pt_3119_b_low.trigger := TRUE;
    ELSE
        pt_3119_b_low.trigger := FALSE;
END_IF
	
//pt_3119-----------------------------------------------------------------------------------------------------
//Instantiate the alarm block, and map the inputs from the OPC GVL
pt_3119_b_high();
pt_3119_b_high.alm_ack:=opc.popa_0082_alarm_ack;
pt_3119_b_high.reset:=opc.popa_0082_alarm_reset;
pt_3119_b_high.priority:=opc.popa_0082_pt_3119_b_high_priority;
pt_3119_b_high.delay_setpoint:=opc.popa_0082_pt_3119_b_high_setpoint;
pt_3119_b_high.enable:=opc.popa_0082_pt_3119_b_high_enable;

//Timer delay elapsed
pt_3119_b_high.delay_ton_et;

//Place your alarm trigger logic here. 
IF io_mapping.pt_3119_b.scaled_value > opc.popa_0082_pt_3119_b_high_setpoint THEN
    pt_3119_b_high.trigger := TRUE;
    ELSE
        pt_3119_b_high.trigger := FALSE;
END_IF
	
//pt_3119-----------------------------------------------------------------------------------------------------
//Instantiate the alarm block, and map the inputs from the OPC GVL
pt_3119_b_high_high();
pt_3119_b_high_high.alm_ack:=opc.popa_0082_alarm_ack;
pt_3119_b_high_high.reset:=opc.popa_0082_alarm_reset;
pt_3119_b_high_high.priority:=opc.popa_0082_pt_3119_b_high_high_priority;
pt_3119_b_high_high.delay_setpoint:=opc.popa_0082_pt_3119_b_high_high_setpoint;
pt_3119_b_high_high.enable:=opc.popa_0082_pt_3119_b_high_high_enable;

//Timer delay elapsed
pt_3119_b_high_high.delay_ton_et;

//Place your alarm trigger logic here. 
IF io_mapping.pt_3119_b.scaled_value >= opc.popa_0082_pt_3119_b_high_high_setpoint THEN
    pt_3119_b_high_high.trigger := TRUE;
    ELSE
        pt_3119_b_high_high.trigger := FALSE;
END_IF


//pt_3219-----------------------------------------------------------------------------------------------------
//Instantiate the alarm block, and map the inputs from the OPC GVL
pt_3219_b_low_low();
pt_3219_b_low_low.alm_ack:=opc.popa_0082_alarm_ack;
pt_3219_b_low_low.reset:=opc.popa_0082_alarm_reset;
pt_3219_b_low_low.priority:=opc.popa_0082_pt_3219_b_low_low_priority;
pt_3219_b_low_low.delay_setpoint:=opc.popa_0082_pt_3219_b_low_low_setpoint;
pt_3219_b_low_low.enable:=opc.popa_0082_pt_3219_b_low_low_enable;

//Timer delay elapsed
pt_3219_b_low_low.delay_ton_et;

//Place your alarm trigger logic here. 
IF io_mapping.pt_3219_b.scaled_value <= opc.popa_0082_pt_3219_b_low_low_setpoint THEN
    pt_3219_b_low_low.trigger := TRUE;
    ELSE
        pt_3219_b_low_low.trigger := FALSE;
END_IF
	
//pt_3219-----------------------------------------------------------------------------------------------------
//Instantiate the alarm block, and map the inputs from the OPC GVL
pt_3219_b_low();
pt_3219_b_low.alm_ack:=opc.popa_0082_alarm_ack;
pt_3219_b_low.reset:=opc.popa_0082_alarm_reset;
pt_3219_b_low.priority:=opc.popa_0082_pt_3219_b_low_priority;
pt_3219_b_low.delay_setpoint:=opc.popa_0082_pt_3219_b_low_setpoint;
pt_3219_b_low.enable:=opc.popa_0082_pt_3219_b_low_enable;

//Timer delay elapsed
pt_3219_b_low.delay_ton_et;

//Place your alarm trigger logic here. 
IF io_mapping.pt_3219_b.scaled_value < opc.popa_0082_pt_3219_b_low_setpoint THEN
    pt_3219_b_low.trigger := TRUE;
    ELSE
        pt_3219_b_low.trigger := FALSE;
END_IF
	
//pt_3219-----------------------------------------------------------------------------------------------------
//Instantiate the alarm block, and map the inputs from the OPC GVL
pt_3219_b_high();
pt_3219_b_high.alm_ack:=opc.popa_0082_alarm_ack;
pt_3219_b_high.reset:=opc.popa_0082_alarm_reset;
pt_3219_b_high.priority:=opc.popa_0082_pt_3219_b_high_priority;
pt_3219_b_high.delay_setpoint:=opc.popa_0082_pt_3219_b_high_setpoint;
pt_3219_b_high.enable:=opc.popa_0082_pt_3219_b_high_enable;

//Timer delay elapsed
pt_3219_b_high.delay_ton_et;

//Place your alarm trigger logic here. 
IF io_mapping.pt_3219_b.scaled_value > opc.popa_0082_pt_3219_b_high_setpoint THEN
    pt_3219_b_high.trigger := TRUE;
    ELSE
        pt_3219_b_high.trigger := FALSE;
END_IF
	
//pt_3219-----------------------------------------------------------------------------------------------------
//Instantiate the alarm block, and map the inputs from the OPC GVL
pt_3219_b_high_high();
pt_3219_b_high_high.alm_ack:=opc.popa_0082_alarm_ack;
pt_3219_b_high_high.reset:=opc.popa_0082_alarm_reset;
pt_3219_b_high_high.priority:=opc.popa_0082_pt_3219_b_high_high_priority;
pt_3219_b_high_high.delay_setpoint:=opc.popa_0082_pt_3219_b_high_high_setpoint;
pt_3219_b_high_high.enable:=opc.popa_0082_pt_3219_b_high_high_enable;

//Timer delay elapsed
pt_3219_b_high_high.delay_ton_et;

//Place your alarm trigger logic here. 
IF io_mapping.pt_3219_b.scaled_value >= opc.popa_0082_pt_3219_b_high_high_setpoint THEN
    pt_3219_b_high_high.trigger := TRUE;
    ELSE
        pt_3219_b_high_high.trigger := FALSE;
END_IF


//pt_3319-----------------------------------------------------------------------------------------------------
//Instantiate the alarm block, and map the inputs from the OPC GVL
pt_3319_b_low_low();
pt_3319_b_low_low.alm_ack:=opc.popa_0082_alarm_ack;
pt_3319_b_low_low.reset:=opc.popa_0082_alarm_reset;
pt_3319_b_low_low.priority:=opc.popa_0082_pt_3319_b_low_low_priority;
pt_3319_b_low_low.delay_setpoint:=opc.popa_0082_pt_3319_b_low_low_setpoint;
pt_3319_b_low_low.enable:=opc.popa_0082_pt_3319_b_low_low_enable;

//Timer delay elapsed
pt_3319_b_low_low.delay_ton_et;

//Place your alarm trigger logic here. 
IF io_mapping.pt_3319_b.scaled_value <= opc.popa_0082_pt_3319_b_low_low_setpoint THEN
    pt_3319_b_low_low.trigger := TRUE;
    ELSE
        pt_3319_b_low_low.trigger := FALSE;
END_IF
	
//pt_3319-----------------------------------------------------------------------------------------------------
//Instantiate the alarm block, and map the inputs from the OPC GVL
pt_3319_b_low();
pt_3319_b_low.alm_ack:=opc.popa_0082_alarm_ack;
pt_3319_b_low.reset:=opc.popa_0082_alarm_reset;
pt_3319_b_low.priority:=opc.popa_0082_pt_3319_b_low_priority;
pt_3319_b_low.delay_setpoint:=opc.popa_0082_pt_3319_b_low_setpoint;
pt_3319_b_low.enable:=opc.popa_0082_pt_3319_b_low_enable;

//Timer delay elapsed
pt_3319_b_low.delay_ton_et;

//Place your alarm trigger logic here. 
IF io_mapping.pt_3319_b.scaled_value < opc.popa_0082_pt_3319_b_low_setpoint THEN
    pt_3319_b_low.trigger := TRUE;
    ELSE
        pt_3319_b_low.trigger := FALSE;
END_IF
	
//pt_3319-----------------------------------------------------------------------------------------------------
//Instantiate the alarm block, and map the inputs from the OPC GVL
pt_3319_b_high();
pt_3319_b_high.alm_ack:=opc.popa_0082_alarm_ack;
pt_3319_b_high.reset:=opc.popa_0082_alarm_reset;
pt_3319_b_high.priority:=opc.popa_0082_pt_3319_b_high_priority;
pt_3319_b_high.delay_setpoint:=opc.popa_0082_pt_3319_b_high_setpoint;
pt_3319_b_high.enable:=opc.popa_0082_pt_3319_b_high_enable;

//Timer delay elapsed
pt_3319_b_high.delay_ton_et;

//Place your alarm trigger logic here. 
IF io_mapping.pt_3319_b.scaled_value > opc.popa_0082_pt_3319_b_high_setpoint THEN
    pt_3319_b_high.trigger := TRUE;
    ELSE
        pt_3319_b_high.trigger := FALSE;
END_IF
	
//pt_3319-----------------------------------------------------------------------------------------------------
//Instantiate the alarm block, and map the inputs from the OPC GVL
pt_3319_b_high_high();
pt_3319_b_high_high.alm_ack:=opc.popa_0082_alarm_ack;
pt_3319_b_high_high.reset:=opc.popa_0082_alarm_reset;
pt_3319_b_high_high.priority:=opc.popa_0082_pt_3319_b_high_high_priority;
pt_3319_b_high_high.delay_setpoint:=opc.popa_0082_pt_3319_b_high_high_setpoint;
pt_3319_b_high_high.enable:=opc.popa_0082_pt_3319_b_high_high_enable;

//Timer delay elapsed
pt_3319_b_high_high.delay_ton_et;

//Place your alarm trigger logic here. 
IF io_mapping.pt_3319_b.scaled_value >= opc.popa_0082_pt_3319_b_high_high_setpoint THEN
    pt_3319_b_high_high.trigger := TRUE;
    ELSE
        pt_3319_b_high_high.trigger := FALSE;
END_IF


//pt_3141-----------------------------------------------------------------------------------------------------
//Instantiate the alarm block, and map the inputs from the OPC GVL
pt_3141_b_low_low();
pt_3141_b_low_low.alm_ack:=opc.popa_0082_alarm_ack;
pt_3141_b_low_low.reset:=opc.popa_0082_alarm_reset;
pt_3141_b_low_low.priority:=opc.popa_0082_pt_3141_b_low_low_priority;
pt_3141_b_low_low.delay_setpoint:=opc.popa_0082_pt_3141_b_low_low_setpoint;
pt_3141_b_low_low.enable:=opc.popa_0082_pt_3141_b_low_low_enable;

//Timer delay elapsed
pt_3141_b_low_low.delay_ton_et;

//Place your alarm trigger logic here. 
IF io_mapping.pt_3141_b.scaled_value <= opc.popa_0082_pt_3141_b_low_low_setpoint THEN
    pt_3141_b_low_low.trigger := TRUE;
    ELSE
        pt_3141_b_low_low.trigger := FALSE;
END_IF
	
//pt_3141-----------------------------------------------------------------------------------------------------
//Instantiate the alarm block, and map the inputs from the OPC GVL
pt_3141_b_low();
pt_3141_b_low.alm_ack:=opc.popa_0082_alarm_ack;
pt_3141_b_low.reset:=opc.popa_0082_alarm_reset;
pt_3141_b_low.priority:=opc.popa_0082_pt_3141_b_low_priority;
pt_3141_b_low.delay_setpoint:=opc.popa_0082_pt_3141_b_low_setpoint;
pt_3141_b_low.enable:=opc.popa_0082_pt_3141_b_low_enable;

//Timer delay elapsed
pt_3141_b_low.delay_ton_et;

//Place your alarm trigger logic here. 
IF io_mapping.pt_3141_b.scaled_value < opc.popa_0082_pt_3141_b_low_setpoint THEN
    pt_3141_b_low.trigger := TRUE;
    ELSE
        pt_3141_b_low.trigger := FALSE;
END_IF
	
//pt_3141-----------------------------------------------------------------------------------------------------
//Instantiate the alarm block, and map the inputs from the OPC GVL
pt_3141_b_high();
pt_3141_b_high.alm_ack:=opc.popa_0082_alarm_ack;
pt_3141_b_high.reset:=opc.popa_0082_alarm_reset;
pt_3141_b_high.priority:=opc.popa_0082_pt_3141_b_high_priority;
pt_3141_b_high.delay_setpoint:=opc.popa_0082_pt_3141_b_high_setpoint;
pt_3141_b_high.enable:=opc.popa_0082_pt_3141_b_high_enable;

//Timer delay elapsed
pt_3141_b_high.delay_ton_et;

//Place your alarm trigger logic here. 
IF io_mapping.pt_3141_b.scaled_value > opc.popa_0082_pt_3141_b_high_setpoint THEN
    pt_3141_b_high.trigger := TRUE;
    ELSE
        pt_3141_b_high.trigger := FALSE;
END_IF
	
//pt_3141-----------------------------------------------------------------------------------------------------
//Instantiate the alarm block, and map the inputs from the OPC GVL
pt_3141_b_high_high();
pt_3141_b_high_high.alm_ack:=opc.popa_0082_alarm_ack;
pt_3141_b_high_high.reset:=opc.popa_0082_alarm_reset;
pt_3141_b_high_high.priority:=opc.popa_0082_pt_3141_b_high_high_priority;
pt_3141_b_high_high.delay_setpoint:=opc.popa_0082_pt_3141_b_high_high_setpoint;
pt_3141_b_high_high.enable:=opc.popa_0082_pt_3141_b_high_high_enable;

//Timer delay elapsed
pt_3141_b_high_high.delay_ton_et;

//Place your alarm trigger logic here. 
IF io_mapping.pt_3141_b.scaled_value >= opc.popa_0082_pt_3141_b_high_high_setpoint THEN
    pt_3141_b_high_high.trigger := TRUE;
    ELSE
        pt_3141_b_high_high.trigger := FALSE;
END_IF


//pt_3241-----------------------------------------------------------------------------------------------------
//Instantiate the alarm block, and map the inputs from the OPC GVL
pt_3241_b_low_low();
pt_3241_b_low_low.alm_ack:=opc.popa_0082_alarm_ack;
pt_3241_b_low_low.reset:=opc.popa_0082_alarm_reset;
pt_3241_b_low_low.priority:=opc.popa_0082_pt_3241_b_low_low_priority;
pt_3241_b_low_low.delay_setpoint:=opc.popa_0082_pt_3241_b_low_low_setpoint;
pt_3241_b_low_low.enable:=opc.popa_0082_pt_3241_b_low_low_enable;

//Timer delay elapsed
pt_3241_b_low_low.delay_ton_et;

//Place your alarm trigger logic here. 
IF io_mapping.pt_3241_b.scaled_value <= opc.popa_0082_pt_3241_b_low_low_setpoint THEN
    pt_3241_b_low_low.trigger := TRUE;
    ELSE
        pt_3241_b_low_low.trigger := FALSE;
END_IF
	
//pt_3241-----------------------------------------------------------------------------------------------------
//Instantiate the alarm block, and map the inputs from the OPC GVL
pt_3241_b_low();
pt_3241_b_low.alm_ack:=opc.popa_0082_alarm_ack;
pt_3241_b_low.reset:=opc.popa_0082_alarm_reset;
pt_3241_b_low.priority:=opc.popa_0082_pt_3241_b_low_priority;
pt_3241_b_low.delay_setpoint:=opc.popa_0082_pt_3241_b_low_setpoint;
pt_3241_b_low.enable:=opc.popa_0082_pt_3241_b_low_enable;

//Timer delay elapsed
pt_3241_b_low.delay_ton_et;

//Place your alarm trigger logic here. 
IF io_mapping.pt_3241_b.scaled_value < opc.popa_0082_pt_3241_b_low_setpoint THEN
    pt_3241_b_low.trigger := TRUE;
    ELSE
        pt_3241_b_low.trigger := FALSE;
END_IF
	
//pt_3241-----------------------------------------------------------------------------------------------------
//Instantiate the alarm block, and map the inputs from the OPC GVL
pt_3241_b_high();
pt_3241_b_high.alm_ack:=opc.popa_0082_alarm_ack;
pt_3241_b_high.reset:=opc.popa_0082_alarm_reset;
pt_3241_b_high.priority:=opc.popa_0082_pt_3241_b_high_priority;
pt_3241_b_high.delay_setpoint:=opc.popa_0082_pt_3241_b_high_setpoint;
pt_3241_b_high.enable:=opc.popa_0082_pt_3241_b_high_enable;

//Timer delay elapsed
pt_3241_b_high.delay_ton_et;

//Place your alarm trigger logic here. 
IF io_mapping.pt_3241_b.scaled_value > opc.popa_0082_pt_3241_b_high_setpoint THEN
    pt_3241_b_high.trigger := TRUE;
    ELSE
        pt_3241_b_high.trigger := FALSE;
END_IF
	
//pt_3241-----------------------------------------------------------------------------------------------------
//Instantiate the alarm block, and map the inputs from the OPC GVL
pt_3241_b_high_high();
pt_3241_b_high_high.alm_ack:=opc.popa_0082_alarm_ack;
pt_3241_b_high_high.reset:=opc.popa_0082_alarm_reset;
pt_3241_b_high_high.priority:=opc.popa_0082_pt_3241_b_high_high_priority;
pt_3241_b_high_high.delay_setpoint:=opc.popa_0082_pt_3241_b_high_high_setpoint;
pt_3241_b_high_high.enable:=opc.popa_0082_pt_3241_b_high_high_enable;

//Timer delay elapsed
pt_3241_b_high_high.delay_ton_et;

//Place your alarm trigger logic here. 
IF io_mapping.pt_3241_b.scaled_value >= opc.popa_0082_pt_3241_b_high_high_setpoint THEN
    pt_3241_b_high_high.trigger := TRUE;
    ELSE
        pt_3241_b_high_high.trigger := FALSE;
END_IF


//pt_3341-----------------------------------------------------------------------------------------------------
//Instantiate the alarm block, and map the inputs from the OPC GVL
pt_3341_b_low_low();
pt_3341_b_low_low.alm_ack:=opc.popa_0082_alarm_ack;
pt_3341_b_low_low.reset:=opc.popa_0082_alarm_reset;
pt_3341_b_low_low.priority:=opc.popa_0082_pt_3341_b_low_low_priority;
pt_3341_b_low_low.delay_setpoint:=opc.popa_0082_pt_3341_b_low_low_setpoint;
pt_3341_b_low_low.enable:=opc.popa_0082_pt_3341_b_low_low_enable;

//Timer delay elapsed
pt_3341_b_low_low.delay_ton_et;

//Place your alarm trigger logic here. 
IF io_mapping.pt_3341_b.scaled_value <= opc.popa_0082_pt_3341_b_low_low_setpoint THEN
    pt_3341_b_low_low.trigger := TRUE;
    ELSE
        pt_3341_b_low_low.trigger := FALSE;
END_IF
	
//pt_3341-----------------------------------------------------------------------------------------------------
//Instantiate the alarm block, and map the inputs from the OPC GVL
pt_3341_b_low();
pt_3341_b_low.alm_ack:=opc.popa_0082_alarm_ack;
pt_3341_b_low.reset:=opc.popa_0082_alarm_reset;
pt_3341_b_low.priority:=opc.popa_0082_pt_3341_b_low_priority;
pt_3341_b_low.delay_setpoint:=opc.popa_0082_pt_3341_b_low_setpoint;
pt_3341_b_low.enable:=opc.popa_0082_pt_3341_b_low_enable;

//Timer delay elapsed
pt_3341_b_low.delay_ton_et;

//Place your alarm trigger logic here. 
IF io_mapping.pt_3341_b.scaled_value < opc.popa_0082_pt_3341_b_low_setpoint THEN
    pt_3341_b_low.trigger := TRUE;
    ELSE
        pt_3341_b_low.trigger := FALSE;
END_IF
	
//pt_3341-----------------------------------------------------------------------------------------------------
//Instantiate the alarm block, and map the inputs from the OPC GVL
pt_3341_b_high();
pt_3341_b_high.alm_ack:=opc.popa_0082_alarm_ack;
pt_3341_b_high.reset:=opc.popa_0082_alarm_reset;
pt_3341_b_high.priority:=opc.popa_0082_pt_3341_b_high_priority;
pt_3341_b_high.delay_setpoint:=opc.popa_0082_pt_3341_b_high_setpoint;
pt_3341_b_high.enable:=opc.popa_0082_pt_3341_b_high_enable;

//Timer delay elapsed
pt_3341_b_high.delay_ton_et;

//Place your alarm trigger logic here. 
IF io_mapping.pt_3341_b.scaled_value > opc.popa_0082_pt_3341_b_high_setpoint THEN
    pt_3341_b_high.trigger := TRUE;
    ELSE
        pt_3341_b_high.trigger := FALSE;
END_IF
	
//pt_3341-----------------------------------------------------------------------------------------------------
//Instantiate the alarm block, and map the inputs from the OPC GVL
pt_3341_b_high_high();
pt_3341_b_high_high.alm_ack:=opc.popa_0082_alarm_ack;
pt_3341_b_high_high.reset:=opc.popa_0082_alarm_reset;
pt_3341_b_high_high.priority:=opc.popa_0082_pt_3341_b_high_high_priority;
pt_3341_b_high_high.delay_setpoint:=opc.popa_0082_pt_3341_b_high_high_setpoint;
pt_3341_b_high_high.enable:=opc.popa_0082_pt_3341_b_high_high_enable;

//Timer delay elapsed
pt_3341_b_high_high.delay_ton_et;

//Place your alarm trigger logic here. 
IF io_mapping.pt_3341_b.scaled_value >= opc.popa_0082_pt_3341_b_high_high_setpoint THEN
    pt_3341_b_high_high.trigger := TRUE;
    ELSE
        pt_3341_b_high_high.trigger := FALSE;
END_IF


//pt_3414-----------------------------------------------------------------------------------------------------
//Instantiate the alarm block, and map the inputs from the OPC GVL
pt_3414_b_low_low();
pt_3414_b_low_low.alm_ack:=opc.popa_0082_alarm_ack;
pt_3414_b_low_low.reset:=opc.popa_0082_alarm_reset;
pt_3414_b_low_low.priority:=opc.popa_0092_pt_3414_b_low_low_priority;
pt_3414_b_low_low.delay_setpoint:=opc.popa_0092_pt_3414_b_low_low_setpoint;
pt_3414_b_low_low.enable:=opc.popa_0092_pt_3414_b_low_low_enable;

//Timer delay elapsed
pt_3414_b_low_low.delay_ton_et;

//Place your alarm trigger logic here. 
IF io_mapping.pt_3414_b.scaled_value <= opc.popa_0092_pt_3414_b_low_low_setpoint THEN
    pt_3414_b_low_low.trigger := TRUE;
    ELSE
        pt_3414_b_low_low.trigger := FALSE;
END_IF
	
//pt_3414-----------------------------------------------------------------------------------------------------
//Instantiate the alarm block, and map the inputs from the OPC GVL
pt_3414_b_low();
pt_3414_b_low.alm_ack:=opc.popa_0082_alarm_ack;
pt_3414_b_low.reset:=opc.popa_0082_alarm_reset;
pt_3414_b_low.priority:=opc.popa_0092_pt_3414_b_low_priority;
pt_3414_b_low.delay_setpoint:=opc.popa_0092_pt_3414_b_low_setpoint;
pt_3414_b_low.enable:=opc.popa_0092_pt_3414_b_low_enable;

//Timer delay elapsed
pt_3414_b_low.delay_ton_et;

//Place your alarm trigger logic here. 
IF io_mapping.pt_3414_b.scaled_value < opc.popa_0092_pt_3414_b_low_setpoint THEN
    pt_3414_b_low.trigger := TRUE;
    ELSE
        pt_3414_b_low.trigger := FALSE;
END_IF
	
//pt_3414-----------------------------------------------------------------------------------------------------
//Instantiate the alarm block, and map the inputs from the OPC GVL
pt_3414_b_high();
pt_3414_b_high.alm_ack:=opc.popa_0082_alarm_ack;
pt_3414_b_high.reset:=opc.popa_0082_alarm_reset;
pt_3414_b_high.priority:=opc.popa_0092_pt_3414_b_high_priority;
pt_3414_b_high.delay_setpoint:=opc.popa_0092_pt_3414_b_high_setpoint;
pt_3414_b_high.enable:=opc.popa_0092_pt_3414_b_high_enable;

//Timer delay elapsed
pt_3414_b_high.delay_ton_et;

//Place your alarm trigger logic here. 
IF io_mapping.pt_3414_b.scaled_value > opc.popa_0092_pt_3414_b_high_setpoint THEN
    pt_3414_b_high.trigger := TRUE;
    ELSE
        pt_3414_b_high.trigger := FALSE;
END_IF
	
//pt_3414-----------------------------------------------------------------------------------------------------
//Instantiate the alarm block, and map the inputs from the OPC GVL
pt_3414_b_high_high();
pt_3414_b_high_high.alm_ack:=opc.popa_0082_alarm_ack;
pt_3414_b_high_high.reset:=opc.popa_0082_alarm_reset;
pt_3414_b_high_high.priority:=opc.popa_0092_pt_3414_b_high_high_priority;
pt_3414_b_high_high.delay_setpoint:=opc.popa_0092_pt_3414_b_high_high_setpoint;
pt_3414_b_high_high.enable:=opc.popa_0092_pt_3414_b_high_high_enable;

//Timer delay elapsed
pt_3414_b_high_high.delay_ton_et;

//Place your alarm trigger logic here. 
IF io_mapping.pt_3414_b.scaled_value >= opc.popa_0092_pt_3414_b_high_high_setpoint THEN
    pt_3414_b_high_high.trigger := TRUE;
    ELSE
        pt_3414_b_high_high.trigger := FALSE;
END_IF

(*

//pt_3428-----------------------------------------------------------------------------------------------------
//Instantiate the alarm block, and map the inputs from the OPC GVL
pt_3428_b_low_low();
pt_3428_b_low_low.alm_ack:=opc.popa_0082_alarm_ack;
pt_3428_b_low_low.reset:=opc.popa_0082_alarm_reset;
pt_3428_b_low_low.priority:=opc.popa_0082_pt_3428_b_low_low_priority;
pt_3428_b_low_low.delay_setpoint:=opc.popa_0082_pt_3428_b_low_low_setpoint;
pt_3428_b_low_low.enable:=opc.popa_0082_pt_3428_b_low_low_enable;

//Timer delay elapsed
pt_3428_b_low_low.delay_ton_et;

//Place your alarm trigger logic here. 
IF io_mapping.pt_3428.scaled_value <= opc.popa_0082_pt_3428_b_low_low_setpoint THEN
    pt_3428_b_low_low.trigger := TRUE;
    ELSE
        pt_3428_b_low_low.trigger := FALSE;
END_IF
	
//pt_3428-----------------------------------------------------------------------------------------------------
//Instantiate the alarm block, and map the inputs from the OPC GVL
pt_3428_b_low();
pt_3428_b_low.alm_ack:=opc.popa_0082_alarm_ack;
pt_3428_b_low.reset:=opc.popa_0082_alarm_reset;
pt_3428_b_low.priority:=opc.popa_0082_pt_3428_b_low_priority;
pt_3428_b_low.delay_setpoint:=opc.popa_0082_pt_3428_b_low_setpoint;
pt_3428_b_low.enable:=opc.popa_0082_pt_3428_b_low_enable;

//Timer delay elapsed
pt_3428_b_low.delay_ton_et;

//Place your alarm trigger logic here. 
IF io_mapping.pt_3428.scaled_value < opc.popa_0082_pt_3428_b_low_setpoint THEN
    pt_3428_b_low.trigger := TRUE;
    ELSE
        pt_3428_b_low.trigger := FALSE;
END_IF
	
//pt_3428-----------------------------------------------------------------------------------------------------
//Instantiate the alarm block, and map the inputs from the OPC GVL
pt_3428_b_high();
pt_3428_b_high.alm_ack:=opc.popa_0082_alarm_ack;
pt_3428_b_high.reset:=opc.popa_0082_alarm_reset;
pt_3428_b_high.priority:=opc.popa_0082_pt_3428_b_high_priority;
pt_3428_b_high.delay_setpoint:=opc.popa_0082_pt_3428_b_high_setpoint;
pt_3428_b_high.enable:=opc.popa_0082_pt_3428_b_high_enable;

//Timer delay elapsed
pt_3428_b_high.delay_ton_et;

//Place your alarm trigger logic here. 
IF io_mapping.pt_3428.scaled_value > opc.popa_0082_pt_3428_b_high_setpoint THEN
    pt_3428_b_high.trigger := TRUE;
    ELSE
        pt_3428_b_high.trigger := FALSE;
END_IF
	
//pt_3428-----------------------------------------------------------------------------------------------------
//Instantiate the alarm block, and map the inputs from the OPC GVL
pt_3428_b_high_high();
pt_3428_b_high_high.alm_ack:=opc.popa_0082_alarm_ack;
pt_3428_b_high_high.reset:=opc.popa_0082_alarm_reset;
pt_3428_b_high_high.priority:=opc.popa_0082_pt_3428_b_high_high_priority;
pt_3428_b_high_high.delay_setpoint:=opc.popa_0082_pt_3428_b_high_high_setpoint;
pt_3428_b_high_high.enable:=opc.popa_0082_pt_3428_b_high_high_enable;

//Timer delay elapsed
pt_3428_b_high_high.delay_ton_et;

//Place your alarm trigger logic here. 
IF io_mapping.pt_3428.scaled_value >= opc.popa_0082_pt_3428_b_high_high_setpoint THEN
    pt_3428_b_high_high.trigger := TRUE;
    ELSE
        pt_3428_b_high_high.trigger := FALSE;
END_IF

*)
//tt_3118-----------------------------------------------------------------------------------------------------
//Instantiate the alarm block, and map the inputs from the OPC GVL
tt_3118_b_low_low();
tt_3118_b_low_low.alm_ack:=opc.popa_0082_alarm_ack;
tt_3118_b_low_low.reset:=opc.popa_0082_alarm_reset;
tt_3118_b_low_low.priority:=opc.popa_0082_tt_3118_b_low_low_priority;
tt_3118_b_low_low.delay_setpoint:=opc.popa_0082_tt_3118_b_low_low_setpoint;
tt_3118_b_low_low.enable:=opc.popa_0082_tt_3118_b_low_low_enable;

//Timer delay elapsed
tt_3118_b_low_low.delay_ton_et;

//Place your alarm trigger logic here. 
IF io_mapping.tt_3118_b.scaled_value <= opc.popa_0082_tt_3118_b_low_low_setpoint THEN
    tt_3118_b_low_low.trigger := TRUE;
    ELSE
        tt_3118_b_low_low.trigger := FALSE;
END_IF
	
//tt_3118-----------------------------------------------------------------------------------------------------
//Instantiate the alarm block, and map the inputs from the OPC GVL
tt_3118_b_low();
tt_3118_b_low.alm_ack:=opc.popa_0082_alarm_ack;
tt_3118_b_low.reset:=opc.popa_0082_alarm_reset;
tt_3118_b_low.priority:=opc.popa_0082_tt_3118_b_low_priority;
tt_3118_b_low.delay_setpoint:=opc.popa_0082_tt_3118_b_low_setpoint;
tt_3118_b_low.enable:=opc.popa_0082_tt_3118_b_low_enable;

//Timer delay elapsed
tt_3118_b_low.delay_ton_et;

//Place your alarm trigger logic here. 
IF io_mapping.tt_3118_b.scaled_value < opc.popa_0082_tt_3118_b_low_setpoint THEN
    tt_3118_b_low.trigger := TRUE;
    ELSE
        tt_3118_b_low.trigger := FALSE;
END_IF
	
//tt_3118-----------------------------------------------------------------------------------------------------
//Instantiate the alarm block, and map the inputs from the OPC GVL
tt_3118_b_high();
tt_3118_b_high.alm_ack:=opc.popa_0082_alarm_ack;
tt_3118_b_high.reset:=opc.popa_0082_alarm_reset;
tt_3118_b_high.priority:=opc.popa_0082_tt_3118_b_high_priority;
tt_3118_b_high.delay_setpoint:=opc.popa_0082_tt_3118_b_high_setpoint;
tt_3118_b_high.enable:=opc.popa_0082_tt_3118_b_high_enable;

//Timer delay elapsed
tt_3118_b_high.delay_ton_et;

//Place your alarm trigger logic here. 
IF io_mapping.tt_3118_b.scaled_value > opc.popa_0082_tt_3118_b_high_setpoint THEN
    tt_3118_b_high.trigger := TRUE;
    ELSE
        tt_3118_b_high.trigger := FALSE;
END_IF
	
//tt_3118-----------------------------------------------------------------------------------------------------
//Instantiate the alarm block, and map the inputs from the OPC GVL
tt_3118_b_high_high();
tt_3118_b_high_high.alm_ack:=opc.popa_0082_alarm_ack;
tt_3118_b_high_high.reset:=opc.popa_0082_alarm_reset;
tt_3118_b_high_high.priority:=opc.popa_0082_tt_3118_b_high_high_priority;
tt_3118_b_high_high.delay_setpoint:=opc.popa_0082_tt_3118_b_high_high_setpoint;
tt_3118_b_high_high.enable:=opc.popa_0082_tt_3118_b_high_high_enable;

//Timer delay elapsed
tt_3118_b_high_high.delay_ton_et;

//Place your alarm trigger logic here. 
IF io_mapping.tt_3118_b.scaled_value >= opc.popa_0082_tt_3118_b_high_high_setpoint THEN
    tt_3118_b_high_high.trigger := TRUE;
    ELSE
        tt_3118_b_high_high.trigger := FALSE;
END_IF


//tt_3218-----------------------------------------------------------------------------------------------------
//Instantiate the alarm block, and map the inputs from the OPC GVL
tt_3218_b_low_low();
tt_3218_b_low_low.alm_ack:=opc.popa_0082_alarm_ack;
tt_3218_b_low_low.reset:=opc.popa_0082_alarm_reset;
tt_3218_b_low_low.priority:=opc.popa_0082_tt_3218_b_low_low_priority;
tt_3218_b_low_low.delay_setpoint:=opc.popa_0082_tt_3218_b_low_low_setpoint;
tt_3218_b_low_low.enable:=opc.popa_0082_tt_3218_b_low_low_enable;

//Timer delay elapsed
tt_3218_b_low_low.delay_ton_et;

//Place your alarm trigger logic here. 
IF io_mapping.tt_3218_b.scaled_value <= opc.popa_0082_tt_3218_b_low_low_setpoint THEN
    tt_3218_b_low_low.trigger := TRUE;
    ELSE
        tt_3218_b_low_low.trigger := FALSE;
END_IF
	
//tt_3218-----------------------------------------------------------------------------------------------------
//Instantiate the alarm block, and map the inputs from the OPC GVL
tt_3218_b_low();
tt_3218_b_low.alm_ack:=opc.popa_0082_alarm_ack;
tt_3218_b_low.reset:=opc.popa_0082_alarm_reset;
tt_3218_b_low.priority:=opc.popa_0082_tt_3218_b_low_priority;
tt_3218_b_low.delay_setpoint:=opc.popa_0082_tt_3218_b_low_setpoint;
tt_3218_b_low.enable:=opc.popa_0082_tt_3218_b_low_enable;

//Timer delay elapsed
tt_3218_b_low.delay_ton_et;

//Place your alarm trigger logic here. 
IF io_mapping.tt_3218_b.scaled_value < opc.popa_0082_tt_3218_b_low_setpoint THEN
    tt_3218_b_low.trigger := TRUE;
    ELSE
        tt_3218_b_low.trigger := FALSE;
END_IF
	
//tt_3218-----------------------------------------------------------------------------------------------------
//Instantiate the alarm block, and map the inputs from the OPC GVL
tt_3218_b_high();
tt_3218_b_high.alm_ack:=opc.popa_0082_alarm_ack;
tt_3218_b_high.reset:=opc.popa_0082_alarm_reset;
tt_3218_b_high.priority:=opc.popa_0082_tt_3218_b_high_priority;
tt_3218_b_high.delay_setpoint:=opc.popa_0082_tt_3218_b_high_setpoint;
tt_3218_b_high.enable:=opc.popa_0082_tt_3218_b_high_enable;

//Timer delay elapsed
tt_3218_b_high.delay_ton_et;

//Place your alarm trigger logic here. 
IF io_mapping.tt_3218_b.scaled_value > opc.popa_0082_tt_3218_b_high_setpoint THEN
    tt_3218_b_high.trigger := TRUE;
    ELSE
        tt_3218_b_high.trigger := FALSE;
END_IF
	
//tt_3218-----------------------------------------------------------------------------------------------------
//Instantiate the alarm block, and map the inputs from the OPC GVL
tt_3218_b_high_high();
tt_3218_b_high_high.alm_ack:=opc.popa_0082_alarm_ack;
tt_3218_b_high_high.reset:=opc.popa_0082_alarm_reset;
tt_3218_b_high_high.priority:=opc.popa_0082_tt_3218_b_high_high_priority;
tt_3218_b_high_high.delay_setpoint:=opc.popa_0082_tt_3218_b_high_high_setpoint;
tt_3218_b_high_high.enable:=opc.popa_0082_tt_3218_b_high_high_enable;

//Timer delay elapsed
tt_3218_b_high_high.delay_ton_et;

//Place your alarm trigger logic here. 
IF io_mapping.tt_3218_b.scaled_value >= opc.popa_0082_tt_3218_b_high_high_setpoint THEN
    tt_3218_b_high_high.trigger := TRUE;
    ELSE
        tt_3218_b_high_high.trigger := FALSE;
END_IF


//tt_3318-----------------------------------------------------------------------------------------------------
//Instantiate the alarm block, and map the inputs from the OPC GVL
tt_3318_b_low_low();
tt_3318_b_low_low.alm_ack:=opc.popa_0082_alarm_ack;
tt_3318_b_low_low.reset:=opc.popa_0082_alarm_reset;
tt_3318_b_low_low.priority:=opc.popa_0082_tt_3318_b_low_low_priority;
tt_3318_b_low_low.delay_setpoint:=opc.popa_0082_tt_3318_b_low_low_setpoint;
tt_3318_b_low_low.enable:=opc.popa_0082_tt_3318_b_low_low_enable;

//Timer delay elapsed
tt_3318_b_low_low.delay_ton_et;

//Place your alarm trigger logic here. 
IF io_mapping.tt_3318_b.scaled_value <= opc.popa_0082_tt_3318_b_low_low_setpoint THEN
    tt_3318_b_low_low.trigger := TRUE;
    ELSE
        tt_3318_b_low_low.trigger := FALSE;
END_IF
	
//tt_3318-----------------------------------------------------------------------------------------------------
//Instantiate the alarm block, and map the inputs from the OPC GVL
tt_3318_b_low();
tt_3318_b_low.alm_ack:=opc.popa_0082_alarm_ack;
tt_3318_b_low.reset:=opc.popa_0082_alarm_reset;
tt_3318_b_low.priority:=opc.popa_0082_tt_3318_b_low_priority;
tt_3318_b_low.delay_setpoint:=opc.popa_0082_tt_3318_b_low_setpoint;
tt_3318_b_low.enable:=opc.popa_0082_tt_3318_b_low_enable;

//Timer delay elapsed
tt_3318_b_low.delay_ton_et;

//Place your alarm trigger logic here. 
IF io_mapping.tt_3318_b.scaled_value < opc.popa_0082_tt_3318_b_low_setpoint THEN
    tt_3318_b_low.trigger := TRUE;
    ELSE
        tt_3318_b_low.trigger := FALSE;
END_IF
	
//tt_3318-----------------------------------------------------------------------------------------------------
//Instantiate the alarm block, and map the inputs from the OPC GVL
tt_3318_b_high();
tt_3318_b_high.alm_ack:=opc.popa_0082_alarm_ack;
tt_3318_b_high.reset:=opc.popa_0082_alarm_reset;
tt_3318_b_high.priority:=opc.popa_0082_tt_3318_b_high_priority;
tt_3318_b_high.delay_setpoint:=opc.popa_0082_tt_3318_b_high_setpoint;
tt_3318_b_high.enable:=opc.popa_0082_tt_3318_b_high_enable;

//Timer delay elapsed
tt_3318_b_high.delay_ton_et;

//Place your alarm trigger logic here. 
IF io_mapping.tt_3318_b.scaled_value > opc.popa_0082_tt_3318_b_high_setpoint THEN
    tt_3318_b_high.trigger := TRUE;
    ELSE
        tt_3318_b_high.trigger := FALSE;
END_IF
	
//tt_3318-----------------------------------------------------------------------------------------------------
//Instantiate the alarm block, and map the inputs from the OPC GVL
tt_3318_b_high_high();
tt_3318_b_high_high.alm_ack:=opc.popa_0082_alarm_ack;
tt_3318_b_high_high.reset:=opc.popa_0082_alarm_reset;
tt_3318_b_high_high.priority:=opc.popa_0082_tt_3318_b_high_high_priority;
tt_3318_b_high_high.delay_setpoint:=opc.popa_0082_tt_3318_b_high_high_setpoint;
tt_3318_b_high_high.enable:=opc.popa_0082_tt_3318_b_high_high_enable;

//Timer delay elapsed
tt_3318_b_high_high.delay_ton_et;

//Place your alarm trigger logic here. 
IF io_mapping.tt_3318_b.scaled_value >= opc.popa_0082_tt_3318_b_high_high_setpoint THEN
    tt_3318_b_high_high.trigger := TRUE;
    ELSE
        tt_3318_b_high_high.trigger := FALSE;
END_IF


//tt_3140-----------------------------------------------------------------------------------------------------
//Instantiate the alarm block, and map the inputs from the OPC GVL
tt_3140_b_low_low();
tt_3140_b_low_low.alm_ack:=opc.popa_0082_alarm_ack;
tt_3140_b_low_low.reset:=opc.popa_0082_alarm_reset;
tt_3140_b_low_low.priority:=opc.popa_0082_tt_3140_b_low_low_priority;
tt_3140_b_low_low.delay_setpoint:=opc.popa_0082_tt_3140_b_low_low_setpoint;
tt_3140_b_low_low.enable:=opc.popa_0082_tt_3140_b_low_low_enable;

//Timer delay elapsed
tt_3140_b_low_low.delay_ton_et;

//Place your alarm trigger logic here. 
IF io_mapping.tt_3140_b.scaled_value <= opc.popa_0082_tt_3140_b_low_low_setpoint THEN
    tt_3140_b_low_low.trigger := TRUE;
    ELSE
        tt_3140_b_low_low.trigger := FALSE;
END_IF
	
//tt_3140-----------------------------------------------------------------------------------------------------
//Instantiate the alarm block, and map the inputs from the OPC GVL
tt_3140_b_low();
tt_3140_b_low.alm_ack:=opc.popa_0082_alarm_ack;
tt_3140_b_low.reset:=opc.popa_0082_alarm_reset;
tt_3140_b_low.priority:=opc.popa_0082_tt_3140_b_low_priority;
tt_3140_b_low.delay_setpoint:=opc.popa_0082_tt_3140_b_low_setpoint;
tt_3140_b_low.enable:=opc.popa_0082_tt_3140_b_low_enable;

//Timer delay elapsed
tt_3140_b_low.delay_ton_et;

//Place your alarm trigger logic here. 
IF io_mapping.tt_3140_b.scaled_value < opc.popa_0082_tt_3140_b_low_setpoint THEN
    tt_3140_b_low.trigger := TRUE;
    ELSE
        tt_3140_b_low.trigger := FALSE;
END_IF
	
//tt_3140-----------------------------------------------------------------------------------------------------
//Instantiate the alarm block, and map the inputs from the OPC GVL
tt_3140_b_high();
tt_3140_b_high.alm_ack:=opc.popa_0082_alarm_ack;
tt_3140_b_high.reset:=opc.popa_0082_alarm_reset;
tt_3140_b_high.priority:=opc.popa_0082_tt_3140_b_high_priority;
tt_3140_b_high.delay_setpoint:=opc.popa_0082_tt_3140_b_high_setpoint;
tt_3140_b_high.enable:=opc.popa_0082_tt_3140_b_high_enable;

//Timer delay elapsed
tt_3140_b_high.delay_ton_et;

//Place your alarm trigger logic here. 
IF io_mapping.tt_3140_b.scaled_value > opc.popa_0082_tt_3140_b_high_setpoint THEN
    tt_3140_b_high.trigger := TRUE;
    ELSE
        tt_3140_b_high.trigger := FALSE;
END_IF
	
//tt_3140-----------------------------------------------------------------------------------------------------
//Instantiate the alarm block, and map the inputs from the OPC GVL
tt_3140_b_high_high();
tt_3140_b_high_high.alm_ack:=opc.popa_0082_alarm_ack;
tt_3140_b_high_high.reset:=opc.popa_0082_alarm_reset;
tt_3140_b_high_high.priority:=opc.popa_0082_tt_3140_b_high_high_priority;
tt_3140_b_high_high.delay_setpoint:=opc.popa_0082_tt_3140_b_high_high_setpoint;
tt_3140_b_high_high.enable:=opc.popa_0082_tt_3140_b_high_high_enable;

//Timer delay elapsed
tt_3140_b_high_high.delay_ton_et;

//Place your alarm trigger logic here. 
IF io_mapping.tt_3140_b.scaled_value >= opc.popa_0082_tt_3140_b_high_high_setpoint THEN
    tt_3140_b_high_high.trigger := TRUE;
    ELSE
        tt_3140_b_high_high.trigger := FALSE;
END_IF


//tt_3240-----------------------------------------------------------------------------------------------------
//Instantiate the alarm block, and map the inputs from the OPC GVL
tt_3240_b_low_low();
tt_3240_b_low_low.alm_ack:=opc.popa_0082_alarm_ack;
tt_3240_b_low_low.reset:=opc.popa_0082_alarm_reset;
tt_3240_b_low_low.priority:=opc.popa_0082_tt_3240_b_low_low_priority;
tt_3240_b_low_low.delay_setpoint:=opc.popa_0082_tt_3240_b_low_low_setpoint;
tt_3240_b_low_low.enable:=opc.popa_0082_tt_3240_b_low_low_enable;

//Timer delay elapsed
tt_3240_b_low_low.delay_ton_et;

//Place your alarm trigger logic here. 
IF io_mapping.tt_3240_b.scaled_value <= opc.popa_0082_tt_3240_b_low_low_setpoint THEN
    tt_3240_b_low_low.trigger := TRUE;
    ELSE
        tt_3240_b_low_low.trigger := FALSE;
END_IF
	
//tt_3240-----------------------------------------------------------------------------------------------------
//Instantiate the alarm block, and map the inputs from the OPC GVL
tt_3240_b_low();
tt_3240_b_low.alm_ack:=opc.popa_0082_alarm_ack;
tt_3240_b_low.reset:=opc.popa_0082_alarm_reset;
tt_3240_b_low.priority:=opc.popa_0082_tt_3240_b_low_priority;
tt_3240_b_low.delay_setpoint:=opc.popa_0082_tt_3240_b_low_setpoint;
tt_3240_b_low.enable:=opc.popa_0082_tt_3240_b_low_enable;

//Timer delay elapsed
tt_3240_b_low.delay_ton_et;

//Place your alarm trigger logic here. 
IF io_mapping.tt_3240_b.scaled_value < opc.popa_0082_tt_3240_b_low_setpoint THEN
    tt_3240_b_low.trigger := TRUE;
    ELSE
        tt_3240_b_low.trigger := FALSE;
END_IF
	
//tt_3240-----------------------------------------------------------------------------------------------------
//Instantiate the alarm block, and map the inputs from the OPC GVL
tt_3240_b_high();
tt_3240_b_high.alm_ack:=opc.popa_0082_alarm_ack;
tt_3240_b_high.reset:=opc.popa_0082_alarm_reset;
tt_3240_b_high.priority:=opc.popa_0082_tt_3240_b_high_priority;
tt_3240_b_high.delay_setpoint:=opc.popa_0082_tt_3240_b_high_setpoint;
tt_3240_b_high.enable:=opc.popa_0082_tt_3240_b_high_enable;

//Timer delay elapsed
tt_3240_b_high.delay_ton_et;

//Place your alarm trigger logic here. 
IF io_mapping.tt_3240_b.scaled_value > opc.popa_0082_tt_3240_b_high_setpoint THEN
    tt_3240_b_high.trigger := TRUE;
    ELSE
        tt_3240_b_high.trigger := FALSE;
END_IF
	
//tt_3240-----------------------------------------------------------------------------------------------------
//Instantiate the alarm block, and map the inputs from the OPC GVL
tt_3240_b_high_high();
tt_3240_b_high_high.alm_ack:=opc.popa_0082_alarm_ack;
tt_3240_b_high_high.reset:=opc.popa_0082_alarm_reset;
tt_3240_b_high_high.priority:=opc.popa_0082_tt_3240_b_high_high_priority;
tt_3240_b_high_high.delay_setpoint:=opc.popa_0082_tt_3240_b_high_high_setpoint;
tt_3240_b_high_high.enable:=opc.popa_0082_tt_3240_b_high_high_enable;

//Timer delay elapsed
tt_3240_b_high_high.delay_ton_et;

//Place your alarm trigger logic here. 
IF io_mapping.tt_3240_b.scaled_value >= opc.popa_0082_tt_3240_b_high_high_setpoint THEN
    tt_3240_b_high_high.trigger := TRUE;
    ELSE
        tt_3240_b_high_high.trigger := FALSE;
END_IF


//tt_3340-----------------------------------------------------------------------------------------------------
//Instantiate the alarm block, and map the inputs from the OPC GVL
tt_3340_b_low_low();
tt_3340_b_low_low.alm_ack:=opc.popa_0082_alarm_ack;
tt_3340_b_low_low.reset:=opc.popa_0082_alarm_reset;
tt_3340_b_low_low.priority:=opc.popa_0082_tt_3340_b_low_low_priority;
tt_3340_b_low_low.delay_setpoint:=opc.popa_0082_tt_3340_b_low_low_setpoint;
tt_3340_b_low_low.enable:=opc.popa_0082_tt_3340_b_low_low_enable;

//Timer delay elapsed
tt_3340_b_low_low.delay_ton_et;

//Place your alarm trigger logic here. 
IF io_mapping.tt_3340_b.scaled_value <= opc.popa_0082_tt_3340_b_low_low_setpoint THEN
    tt_3340_b_low_low.trigger := TRUE;
    ELSE
        tt_3340_b_low_low.trigger := FALSE;
END_IF
	
//tt_3340-----------------------------------------------------------------------------------------------------
//Instantiate the alarm block, and map the inputs from the OPC GVL
tt_3340_b_low();
tt_3340_b_low.alm_ack:=opc.popa_0082_alarm_ack;
tt_3340_b_low.reset:=opc.popa_0082_alarm_reset;
tt_3340_b_low.priority:=opc.popa_0082_tt_3340_b_low_priority;
tt_3340_b_low.delay_setpoint:=opc.popa_0082_tt_3340_b_low_setpoint;
tt_3340_b_low.enable:=opc.popa_0082_tt_3340_b_low_enable;

//Timer delay elapsed
tt_3340_b_low.delay_ton_et;

//Place your alarm trigger logic here. 
IF io_mapping.tt_3340_b.scaled_value < opc.popa_0082_tt_3340_b_low_setpoint THEN
    tt_3340_b_low.trigger := TRUE;
    ELSE
        tt_3340_b_low.trigger := FALSE;
END_IF
	
//tt_3340-----------------------------------------------------------------------------------------------------
//Instantiate the alarm block, and map the inputs from the OPC GVL
tt_3340_b_high();
tt_3340_b_high.alm_ack:=opc.popa_0082_alarm_ack;
tt_3340_b_high.reset:=opc.popa_0082_alarm_reset;
tt_3340_b_high.priority:=opc.popa_0082_tt_3340_b_high_priority;
tt_3340_b_high.delay_setpoint:=opc.popa_0082_tt_3340_b_high_setpoint;
tt_3340_b_high.enable:=opc.popa_0082_tt_3340_b_high_enable;

//Timer delay elapsed
tt_3340_b_high.delay_ton_et;

//Place your alarm trigger logic here. 
IF io_mapping.tt_3340_b.scaled_value > opc.popa_0082_tt_3340_b_high_setpoint THEN
    tt_3340_b_high.trigger := TRUE;
    ELSE
        tt_3340_b_high.trigger := FALSE;
END_IF
	
//tt_3340-----------------------------------------------------------------------------------------------------
//Instantiate the alarm block, and map the inputs from the OPC GVL
tt_3340_b_high_high();
tt_3340_b_high_high.alm_ack:=opc.popa_0082_alarm_ack;
tt_3340_b_high_high.reset:=opc.popa_0082_alarm_reset;
tt_3340_b_high_high.priority:=opc.popa_0082_tt_3340_b_high_high_priority;
tt_3340_b_high_high.delay_setpoint:=opc.popa_0082_tt_3340_b_high_high_setpoint;
tt_3340_b_high_high.enable:=opc.popa_0082_tt_3340_b_high_high_enable;

//Timer delay elapsed
tt_3340_b_high_high.delay_ton_et;

//Place your alarm trigger logic here. 
IF io_mapping.tt_3340_b.scaled_value >= opc.popa_0082_tt_3340_b_high_high_setpoint THEN
    tt_3340_b_high_high.trigger := TRUE;
    ELSE
        tt_3340_b_high_high.trigger := FALSE;
END_IF


//tt_3432-----------------------------------------------------------------------------------------------------
//Instantiate the alarm block, and map the inputs from the OPC GVL
tt_3432_b_low_low();
tt_3432_b_low_low.alm_ack:=opc.popa_0082_alarm_ack;
tt_3432_b_low_low.reset:=opc.popa_0082_alarm_reset;
tt_3432_b_low_low.priority:=opc.popa_0092_tt_3432_b_low_low_priority;
tt_3432_b_low_low.delay_setpoint:=opc.popa_0092_tt_3432_b_low_low_setpoint;
tt_3432_b_low_low.enable:=opc.popa_0092_tt_3432_b_low_low_enable;

//Timer delay elapsed
tt_3432_b_low_low.delay_ton_et;

//Place your alarm trigger logic here. 
IF io_mapping.tt_3432_b.scaled_value <= opc.popa_0092_tt_3432_b_low_low_setpoint THEN
    tt_3432_b_low_low.trigger := TRUE;
    ELSE
        tt_3432_b_low_low.trigger := FALSE;
END_IF
	
//tt_3432-----------------------------------------------------------------------------------------------------
//Instantiate the alarm block, and map the inputs from the OPC GVL
tt_3432_b_low();
tt_3432_b_low.alm_ack:=opc.popa_0082_alarm_ack;
tt_3432_b_low.reset:=opc.popa_0082_alarm_reset;
tt_3432_b_low.priority:=opc.popa_0092_tt_3432_b_low_priority;
tt_3432_b_low.delay_setpoint:=opc.popa_0092_tt_3432_b_low_setpoint;
tt_3432_b_low.enable:=opc.popa_0092_tt_3432_b_low_enable;

//Timer delay elapsed
tt_3432_b_low.delay_ton_et;

//Place your alarm trigger logic here. 
IF io_mapping.tt_3432_b.scaled_value < opc.popa_0092_tt_3432_b_low_setpoint THEN
    tt_3432_b_low.trigger := TRUE;
    ELSE
        tt_3432_b_low.trigger := FALSE;
END_IF
	
//tt_3432-----------------------------------------------------------------------------------------------------
//Instantiate the alarm block, and map the inputs from the OPC GVL
tt_3432_b_high();
tt_3432_b_high.alm_ack:=opc.popa_0082_alarm_ack;
tt_3432_b_high.reset:=opc.popa_0082_alarm_reset;
tt_3432_b_high.priority:=opc.popa_0092_tt_3432_b_high_priority;
tt_3432_b_high.delay_setpoint:=opc.popa_0092_tt_3432_b_high_setpoint;
tt_3432_b_high.enable:=opc.popa_0092_tt_3432_b_high_enable;

//Timer delay elapsed
tt_3432_b_high.delay_ton_et;

//Place your alarm trigger logic here. 
IF io_mapping.tt_3432_b.scaled_value > opc.popa_0092_tt_3432_b_high_setpoint THEN
    tt_3432_b_high.trigger := TRUE;
    ELSE
        tt_3432_b_high.trigger := FALSE;
END_IF
	
//tt_3432-----------------------------------------------------------------------------------------------------
//Instantiate the alarm block, and map the inputs from the OPC GVL
tt_3432_b_high_high();
tt_3432_b_high_high.alm_ack:=opc.popa_0082_alarm_ack;
tt_3432_b_high_high.reset:=opc.popa_0082_alarm_reset;
tt_3432_b_high_high.priority:=opc.popa_0092_tt_3432_b_high_high_priority;
tt_3432_b_high_high.delay_setpoint:=opc.popa_0092_tt_3432_b_high_high_setpoint;
tt_3432_b_high_high.enable:=opc.popa_0092_tt_3432_b_high_high_enable;

//Timer delay elapsed
tt_3432_b_high_high.delay_ton_et;

//Place your alarm trigger logic here. 
IF io_mapping.tt_3432_b.scaled_value >= opc.popa_0092_tt_3432_b_high_high_setpoint THEN
    tt_3432_b_high_high.trigger := TRUE;
    ELSE
        tt_3432_b_high_high.trigger := FALSE;
END_IF

END_PROGRAM

// ---- POUs/Function Blocks/alarm.TcPOU
FUNCTION_BLOCK alarm
VAR_INPUT
	//Input that triggers the alarm condition
	trigger : BOOL;
	//Alarm Acknowledge bit, Clears low priority alarms
	alm_ack : BOOL;
	//Alarm Reset, clears high priority alarms
	reset : BOOL;
	//Alarm Priority, 1=Warning, 2=Error, 3=Critical
	priority : INT;
	//Alarm Delay Setpoint in Seconds
	delay_setpoint : REAL;
	//Alarm Enable
	enable : BOOL;
END_VAR
VAR_OUTPUT
	//Alarm is triggered
	active : BOOL;
	delay_ton_et : TIME;
END_VAR
VAR
	//Delay Timer Tags
	delay_ton : TON;
	delay_ton_pt : TIME;
	//delay_ton_et : TIME;
	//Delay setpoint converted to Milliseconds
	delay_ms : REAL;
	//Cutoff for needing to reset vs ack an alarm.  At or above this value requires reset.  
	reset_priority : REAL :=3;
END_VAR

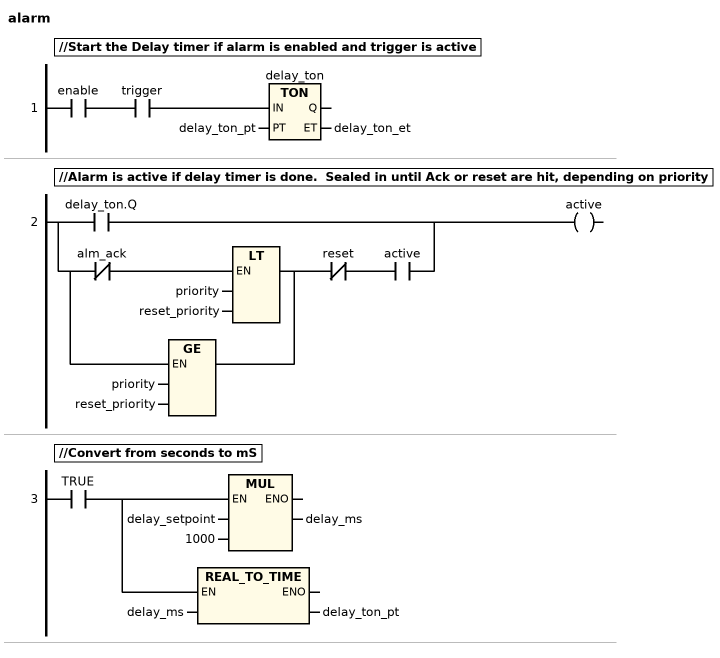
// NETWORK 1
// label: //Start the Delay timer if alarm is enabled and trigger is active
delay_ton(IN := enable AND trigger, PT := delay_ton_pt, ET => delay_ton_et); // TON

// NETWORK 2
// label: //Alarm is active if delay timer is done.  Sealed in until Ack or reset are hit, depending on priority
active := delay_ton.Q OR (NOT alm_ack AND priority < reset_priority OR priority >= reset_priority) AND NOT reset AND active;

// NETWORK 3
// label: //Convert from seconds to mS
delay_ms := delay_setpoint * 1000;
delay_ton_pt := REAL_TO_TIME(delay_ms);

END_FUNCTION_BLOCK

// ---- POUs/pump_manager.TcPOU
PROGRAM pump_manager
VAR
	//Repeat for each pump?
	u_3112_b : motor_vfd;
	u_3112_b_pid : FB_BasicPID;
	u_3112_b_pid_error : UINT;
	u_3112_b_pid_output : REAL;
	u_3112_b_enable: BOOL;
	u_3112_b_idle_request: BOOL;
	u_3112_b_cip_request: BOOL;
	u_3112_b_manual_request: BOOL;
	u_3112_b_stop_request: BOOL;
	u_3112_b_intlk: BOOL;
	u_3112_b_maint_request: BOOL;
	u_3112_b_idle_speed_request: REAL;
	u_3112_b_setpoint_request: REAL;
	u_3112_b_cip_speed_request: REAL;
	u_3112_b_manual_speed_request: REAL;
	u_3112_b_maint_speed_request: REAL;
	
	u_3212_b : motor_vfd;
	u_3212_b_pid : FB_BasicPID;
	u_3212_b_pid_error : UINT;
	u_3212_b_enable: BOOL;
	u_3212_b_idle_request: BOOL;
	u_3212_b_cip_request: BOOL;
	u_3212_b_manual_request: BOOL;
	u_3212_b_stop_request: BOOL;
	u_3212_b_intlk: BOOL;
	u_3212_b_maint_request: BOOL;
	u_3212_b_idle_speed_request: REAL;
	u_3212_b_setpoint_request: REAL;
	u_3212_b_cip_speed_request: REAL;
	u_3212_b_manual_speed_request: REAL;
	u_3212_b_maint_speed_request: REAL;
	
	u_3312_b : motor_vfd;
	u_3312_b_pid : FB_BasicPID;
	u_3312_b_pid_error : UINT;
	u_3312_b_enable: BOOL;
	u_3312_b_idle_request: BOOL;
	u_3312_b_cip_request: BOOL;
	u_3312_b_manual_request: BOOL;
	u_3312_b_stop_request: BOOL;
	u_3312_b_intlk: BOOL;
	u_3312_b_maint_request: BOOL;
	u_3312_b_idle_speed_request: REAL;
	u_3312_b_speed_request: REAL;
	u_3312_b_cip_speed_request: REAL;
	u_3312_b_manual_speed_request: REAL;
	u_3312_b_maint_speed_request: REAL;
	
	u_3405_b : motor_vfd;
	u_3405_b_pid : FB_BasicPID;
	u_3405_b_pid_error : UINT;
	u_3405_b_enable: BOOL;
	u_3405_b_idle_request: BOOL;
	u_3405_b_cip_request: BOOL;
	u_3405_b_manual_request: BOOL;
	u_3405_b_stop_request: BOOL;
	u_3405_b_intlk: BOOL;
	u_3405_b_maint_request: BOOL;
	u_3405_b_idle_speed_request: REAL;
	u_3405_b_speed_request: REAL;
	u_3405_b_cip_speed_request: REAL;
	u_3405_b_manual_speed_request: REAL;
	u_3405_b_maint_speed_request: REAL;
	
	u_3160_b : motor_vfd;
	u_3160_b_pid : FB_BasicPID;
	u_3160_b_pid_error : UINT;
	u_3160_b_enable: BOOL;
	u_3160_b_idle_request: BOOL;
	u_3160_b_cip_request: BOOL;
	u_3160_b_manual_request: BOOL;
	u_3160_b_stop_request: BOOL;
	u_3160_b_intlk: BOOL;
	u_3160_b_maint_request: BOOL;
	u_3160_b_idle_speed_request: REAL;
	u_3160_b_speed_request: REAL;
	u_3160_b_cip_speed_request: REAL;
	u_3160_b_manual_speed_request: REAL;
	u_3160_b_maint_speed_request: REAL;
	
	u_3260_b : motor_vfd;
	u_3260_b_pid : FB_BasicPID;
	u_3260_b_pid_error : UINT;
	u_3260_b_enable: BOOL;
	u_3260_b_idle_request: BOOL;
	u_3260_b_cip_request: BOOL;
	u_3260_b_manual_request: BOOL;
	u_3260_b_stop_request: BOOL;
	u_3260_b_intlk: BOOL;
	u_3260_b_maint_request: BOOL;
	u_3260_b_idle_speed_request: REAL;
	u_3260_b_speed_request: REAL;
	u_3260_b_cip_speed_request: REAL;
	u_3260_b_manual_speed_request: REAL;
	u_3260_b_maint_speed_request: REAL;
	
	u_3360_b : motor_vfd;
	u_3360_b_pid : FB_BasicPID;
	u_3360_b_pid_error : UINT;
	u_3360_b_enable: BOOL;
	u_3360_b_idle_request: BOOL;
	u_3360_b_cip_request: BOOL;
	u_3360_b_manual_request: BOOL;
	u_3360_b_stop_request: BOOL;
	u_3360_b_intlk: BOOL;
	u_3360_b_maint_request: BOOL;
	u_3360_b_idle_speed_request: REAL;
	u_3360_b_speed_request: REAL;
	u_3360_b_cip_speed_request: REAL;
	u_3360_b_manual_speed_request: REAL;
	u_3360_b_maint_speed_request: REAL;
	
	
	gen_alm_active: BOOL;
	ed_routine_idle: BOOL;
	ed_routine_cip: BOOL;
	//ed_routine_manual: BOOL;
	ed_routine_maint: BOOL;
	
	u_3370_b : motor_vfd;
	u_3370_b_pid : FB_BasicPID;
	u_3370_b_pid_error : UINT;
	u_3370_b_enable: BOOL;
	u_3370_b_idle_request: BOOL;
	u_3370_b_cip_request: BOOL;
	u_3370_b_manual_request: BOOL;
	u_3370_b_stop_request: BOOL;
	u_3370_b_intlk: BOOL;
	u_3370_b_maint_request: BOOL;
	u_3370_b_idle_speed_request: REAL;
	u_3370_b_speed_request: REAL;
	u_3370_b_cip_speed_request: REAL;
	u_3370_b_manual_speed_request: REAL;
	u_3370_b_maint_speed_request: REAL;
	u_3312_b_setpoint_request: REAL;
	u_3405_b_setpoint_request: REAL;
	
	u_3112_b_pid_reset: BOOL;
	u_3112_b_ons: R_TRIG;
	u_3312_b_pid_reset: BOOL;
	u_3312_b_ons: R_TRIG;
	u_3212_b_ons: R_TRIG;
	u_3212_b_pid_reset: BOOL;
	u_3405_b_ons: R_TRIG;
	u_3405_b_pid_reset: BOOL;
	u_3370_b_setpoint_request: REAL;
	u_3370_b_ons: R_TRIG;
	u_3370_b_pid_reset: BOOL;
	u_3112_b_speed_request: REAL;
	u_3212_b_speed_request: REAL;
END_VAR
VAR // added by the converter: edge detectors and wires of the graphical bodies
    _w1, _w2, _w3, _w4, _w5, _w6, _w7, _w8, _w9, _w10, _w11, _w12, _w13, _w14, _w15, _w16, _w17, _w18, _w19, _w20, _w21, _w22, _w23, _w24, _w25, _w26, _w27, _w28 : BOOL;
END_VAR

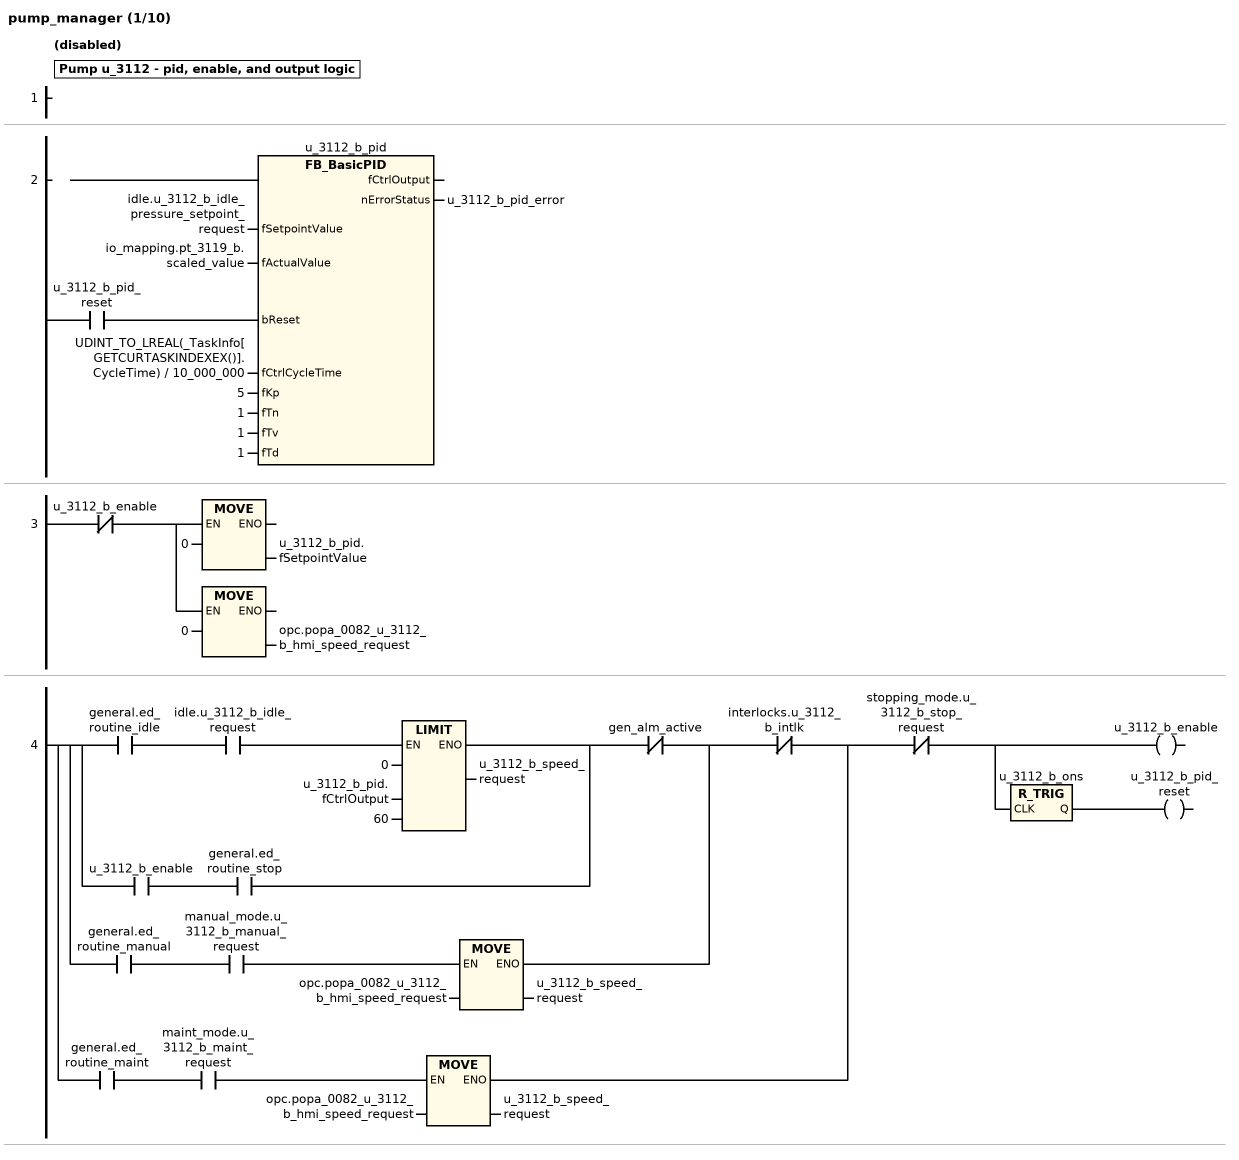
// NETWORK 1 (disabled)
// label: Pump u_3112 - pid, enable, and output logic

// NETWORK 2
u_3112_b_pid(
    fSetpointValue := idle.u_3112_b_idle_pressure_setpoint_request,
    fActualValue := io_mapping.pt_3119_b.scaled_value,
    bReset := u_3112_b_pid_reset,
    fCtrlCycleTime := UDINT_TO_LREAL(_TaskInfo[GETCURTASKINDEXEX()].CycleTime) / 10_000_000,
    fKp := 5,
    fTn := 1,
    fTv := 1,
    fTd := 1,
    nErrorStatus => u_3112_b_pid_error); // FB_BasicPID

// NETWORK 3
_w1 := NOT u_3112_b_enable;
IF _w1 THEN u_3112_b_pid.fSetpointValue := 0; END_IF
IF _w1 THEN opc.popa_0082_u_3112_b_hmi_speed_request := 0; END_IF

// NETWORK 4
_w2 := general.ed_routine_idle AND idle.u_3112_b_idle_request;
IF _w2 THEN u_3112_b_speed_request := LIMIT(0, u_3112_b_pid.fCtrlOutput, 60); END_IF
_w3 := general.ed_routine_manual AND manual_mode.u_3112_b_manual_request;
IF _w3 THEN u_3112_b_speed_request := opc.popa_0082_u_3112_b_hmi_speed_request; END_IF
_w4 := general.ed_routine_maint AND maint_mode.u_3112_b_maint_request;
IF _w4 THEN u_3112_b_speed_request := opc.popa_0082_u_3112_b_hmi_speed_request; END_IF
_w5 := (((_w2 OR u_3112_b_enable AND general.ed_routine_stop) AND NOT gen_alm_active OR _w3) AND NOT interlocks.u_3112_b_intlk OR _w4) AND NOT stopping_mode.u_3112_b_stop_request;
u_3112_b_enable := _w5;
u_3112_b_ons(CLK := _w5); // R_TRIG
u_3112_b_pid_reset := u_3112_b_ons.Q;

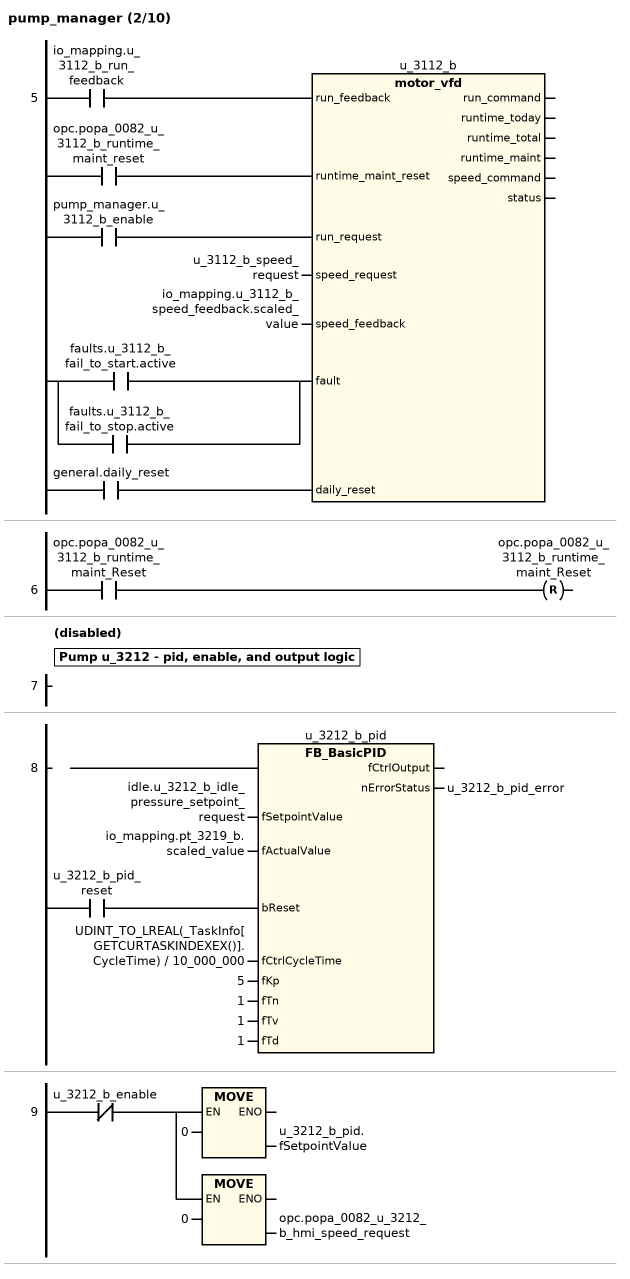
// NETWORK 5
u_3112_b(
    run_feedback := io_mapping.u_3112_b_run_feedback,
    runtime_maint_reset := opc.popa_0082_u_3112_b_runtime_maint_reset,
    run_request := pump_manager.u_3112_b_enable,
    speed_request := u_3112_b_speed_request,
    speed_feedback := io_mapping.u_3112_b_speed_feedback.scaled_value,
    fault := faults.u_3112_b_fail_to_start.active OR faults.u_3112_b_fail_to_stop.active,
    daily_reset := general.daily_reset); // motor_vfd

// NETWORK 6
opc.popa_0082_u_3112_b_runtime_maint_Reset R= opc.popa_0082_u_3112_b_runtime_maint_Reset;

// NETWORK 7 (disabled)
// label: Pump u_3212 - pid, enable, and output logic

// NETWORK 8
u_3212_b_pid(
    fSetpointValue := idle.u_3212_b_idle_pressure_setpoint_request,
    fActualValue := io_mapping.pt_3219_b.scaled_value,
    bReset := u_3212_b_pid_reset,
    fCtrlCycleTime := UDINT_TO_LREAL(_TaskInfo[GETCURTASKINDEXEX()].CycleTime) / 10_000_000,
    fKp := 5,
    fTn := 1,
    fTv := 1,
    fTd := 1,
    nErrorStatus => u_3212_b_pid_error); // FB_BasicPID

// NETWORK 9
_w6 := NOT u_3212_b_enable;
IF _w6 THEN u_3212_b_pid.fSetpointValue := 0; END_IF
IF _w6 THEN opc.popa_0082_u_3212_b_hmi_speed_request := 0; END_IF

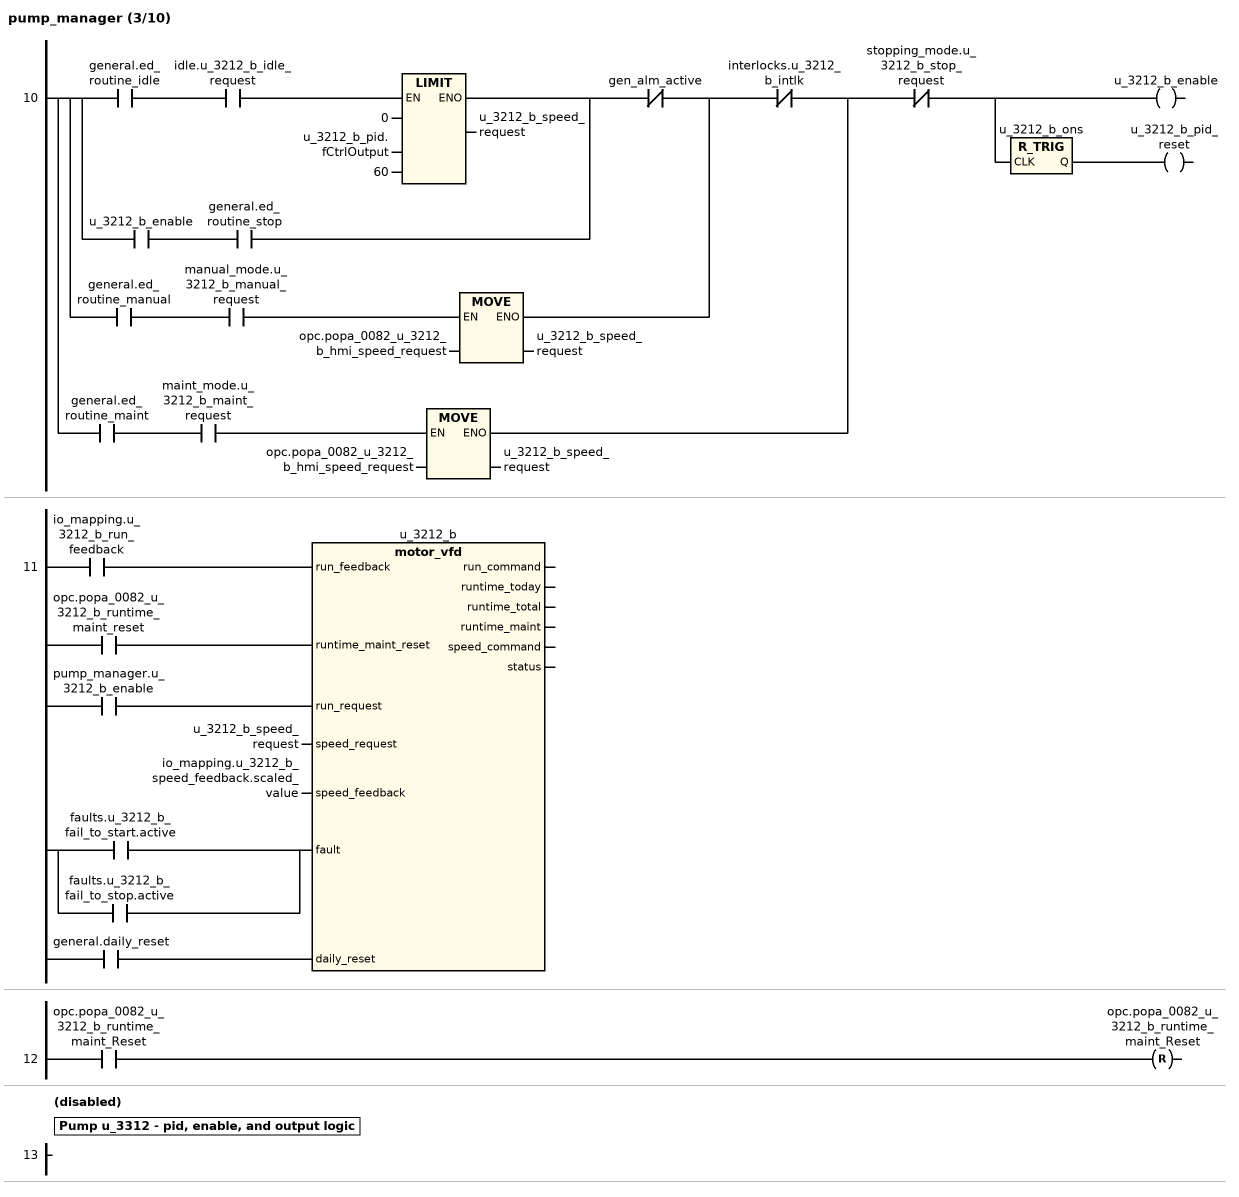
// NETWORK 10
_w7 := general.ed_routine_idle AND idle.u_3212_b_idle_request;
IF _w7 THEN u_3212_b_speed_request := LIMIT(0, u_3212_b_pid.fCtrlOutput, 60); END_IF
_w8 := general.ed_routine_manual AND manual_mode.u_3212_b_manual_request;
IF _w8 THEN u_3212_b_speed_request := opc.popa_0082_u_3212_b_hmi_speed_request; END_IF
_w9 := general.ed_routine_maint AND maint_mode.u_3212_b_maint_request;
IF _w9 THEN u_3212_b_speed_request := opc.popa_0082_u_3212_b_hmi_speed_request; END_IF
_w10 := (((_w7 OR u_3212_b_enable AND general.ed_routine_stop) AND NOT gen_alm_active OR _w8) AND NOT interlocks.u_3212_b_intlk OR _w9) AND NOT stopping_mode.u_3212_b_stop_request;
u_3212_b_enable := _w10;
u_3212_b_ons(CLK := _w10); // R_TRIG
u_3212_b_pid_reset := u_3212_b_ons.Q;

// NETWORK 11
u_3212_b(
    run_feedback := io_mapping.u_3212_b_run_feedback,
    runtime_maint_reset := opc.popa_0082_u_3212_b_runtime_maint_reset,
    run_request := pump_manager.u_3212_b_enable,
    speed_request := u_3212_b_speed_request,
    speed_feedback := io_mapping.u_3212_b_speed_feedback.scaled_value,
    fault := faults.u_3212_b_fail_to_start.active OR faults.u_3212_b_fail_to_stop.active,
    daily_reset := general.daily_reset); // motor_vfd

// NETWORK 12
opc.popa_0082_u_3212_b_runtime_maint_Reset R= opc.popa_0082_u_3212_b_runtime_maint_Reset;

// NETWORK 13 (disabled)
// label: Pump u_3312 - pid, enable, and output logic

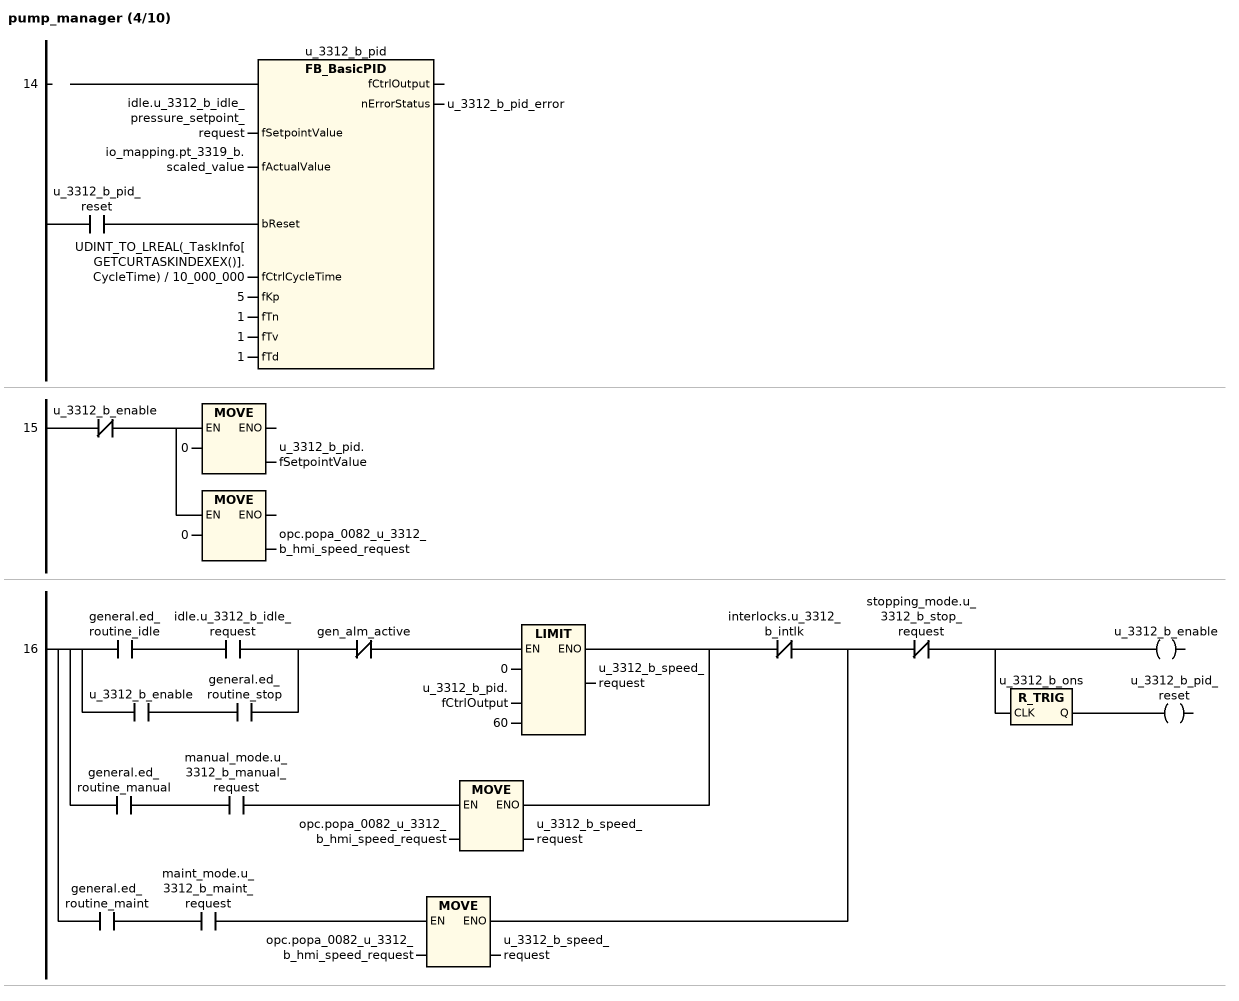
// NETWORK 14
u_3312_b_pid(
    fSetpointValue := idle.u_3312_b_idle_pressure_setpoint_request,
    fActualValue := io_mapping.pt_3319_b.scaled_value,
    bReset := u_3312_b_pid_reset,
    fCtrlCycleTime := UDINT_TO_LREAL(_TaskInfo[GETCURTASKINDEXEX()].CycleTime) / 10_000_000,
    fKp := 5,
    fTn := 1,
    fTv := 1,
    fTd := 1,
    nErrorStatus => u_3312_b_pid_error); // FB_BasicPID

// NETWORK 15
_w11 := NOT u_3312_b_enable;
IF _w11 THEN u_3312_b_pid.fSetpointValue := 0; END_IF
IF _w11 THEN opc.popa_0082_u_3312_b_hmi_speed_request := 0; END_IF

// NETWORK 16
_w12 := (general.ed_routine_idle AND idle.u_3312_b_idle_request OR u_3312_b_enable AND general.ed_routine_stop) AND NOT gen_alm_active;
IF _w12 THEN u_3312_b_speed_request := LIMIT(0, u_3312_b_pid.fCtrlOutput, 60); END_IF
_w13 := general.ed_routine_manual AND manual_mode.u_3312_b_manual_request;
IF _w13 THEN u_3312_b_speed_request := opc.popa_0082_u_3312_b_hmi_speed_request; END_IF
_w14 := general.ed_routine_maint AND maint_mode.u_3312_b_maint_request;
IF _w14 THEN u_3312_b_speed_request := opc.popa_0082_u_3312_b_hmi_speed_request; END_IF
_w15 := ((_w12 OR _w13) AND NOT interlocks.u_3312_b_intlk OR _w14) AND NOT stopping_mode.u_3312_b_stop_request;
u_3312_b_enable := _w15;
u_3312_b_ons(CLK := _w15); // R_TRIG
u_3312_b_pid_reset := u_3312_b_ons.Q;

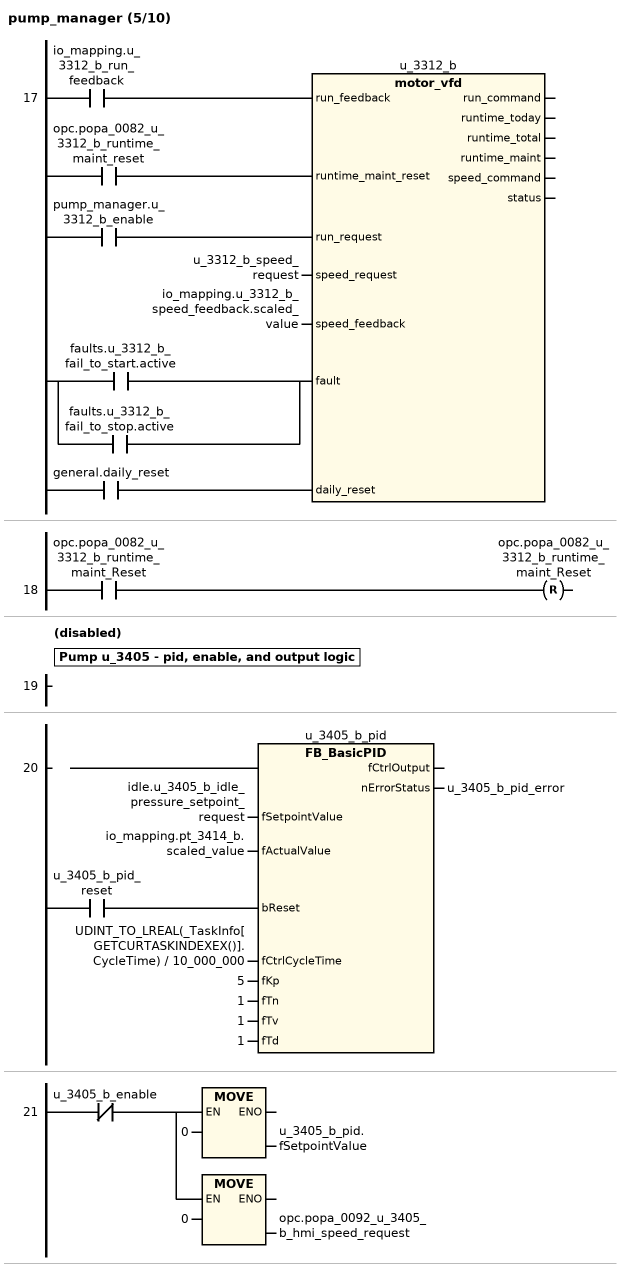
// NETWORK 17
u_3312_b(
    run_feedback := io_mapping.u_3312_b_run_feedback,
    runtime_maint_reset := opc.popa_0082_u_3312_b_runtime_maint_reset,
    run_request := pump_manager.u_3312_b_enable,
    speed_request := u_3312_b_speed_request,
    speed_feedback := io_mapping.u_3312_b_speed_feedback.scaled_value,
    fault := faults.u_3312_b_fail_to_start.active OR faults.u_3312_b_fail_to_stop.active,
    daily_reset := general.daily_reset); // motor_vfd

// NETWORK 18
opc.popa_0082_u_3312_b_runtime_maint_Reset R= opc.popa_0082_u_3312_b_runtime_maint_Reset;

// NETWORK 19 (disabled)
// label: Pump u_3405 - pid, enable, and output logic

// NETWORK 20
u_3405_b_pid(
    fSetpointValue := idle.u_3405_b_idle_pressure_setpoint_request,
    fActualValue := io_mapping.pt_3414_b.scaled_value,
    bReset := u_3405_b_pid_reset,
    fCtrlCycleTime := UDINT_TO_LREAL(_TaskInfo[GETCURTASKINDEXEX()].CycleTime) / 10_000_000,
    fKp := 5,
    fTn := 1,
    fTv := 1,
    fTd := 1,
    nErrorStatus => u_3405_b_pid_error); // FB_BasicPID

// NETWORK 21
_w16 := NOT u_3405_b_enable;
IF _w16 THEN u_3405_b_pid.fSetpointValue := 0; END_IF
IF _w16 THEN opc.popa_0092_u_3405_b_hmi_speed_request := 0; END_IF

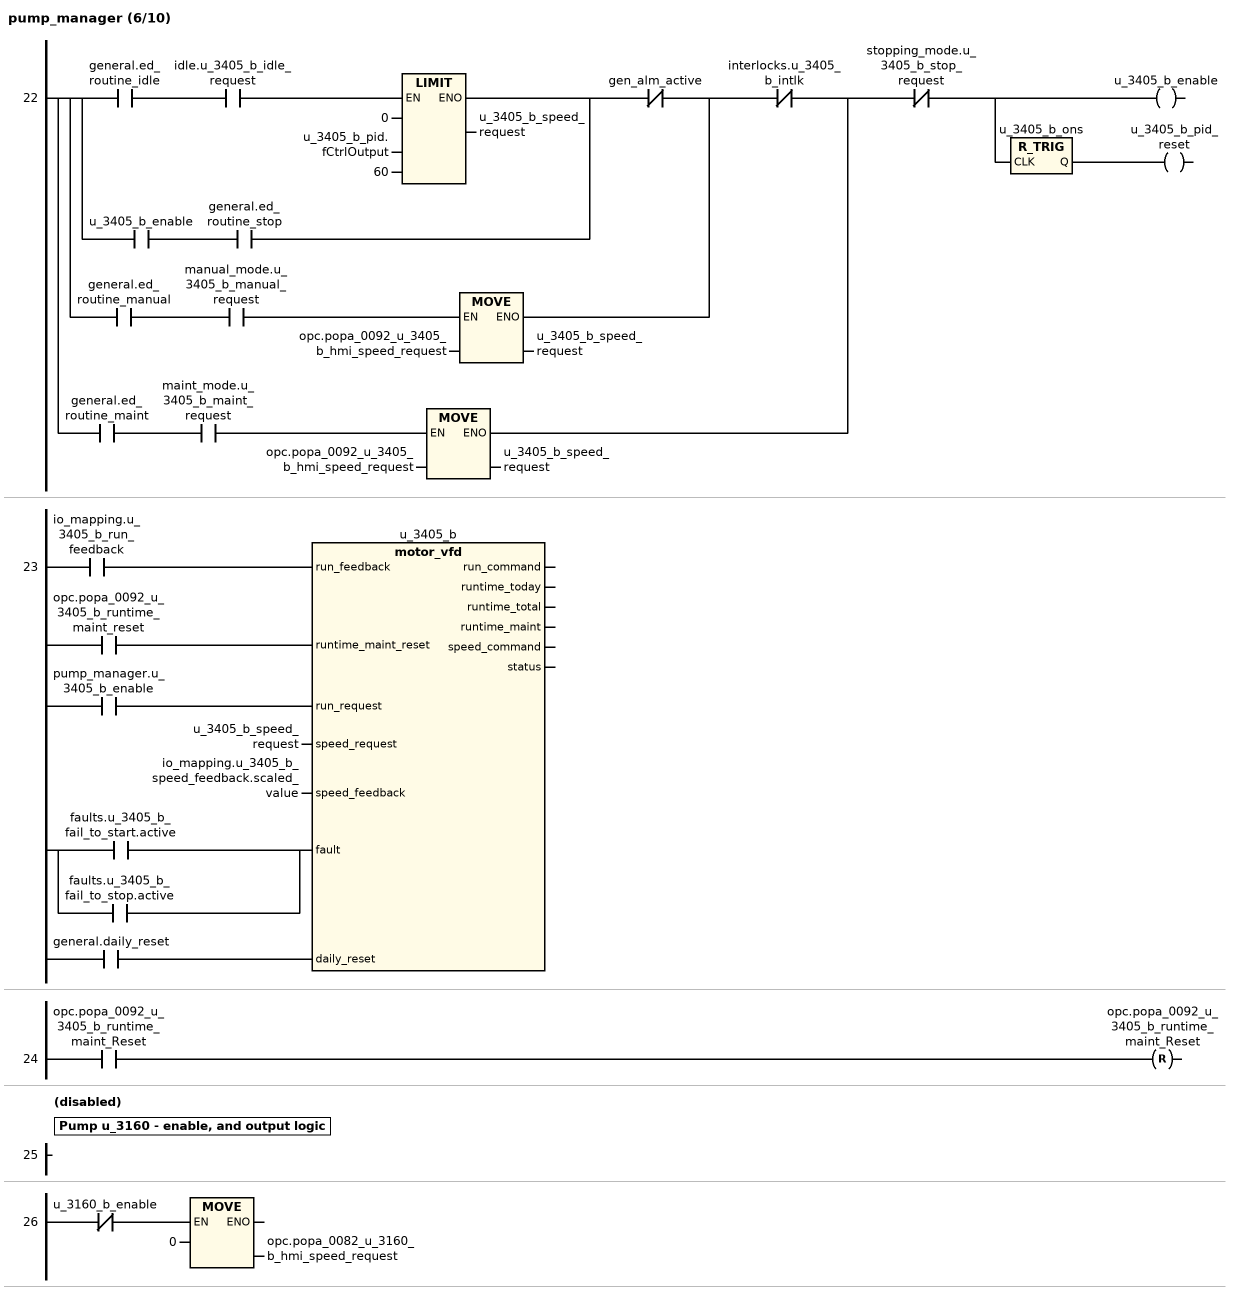
// NETWORK 22
_w17 := general.ed_routine_idle AND idle.u_3405_b_idle_request;
IF _w17 THEN u_3405_b_speed_request := LIMIT(0, u_3405_b_pid.fCtrlOutput, 60); END_IF
_w18 := general.ed_routine_manual AND manual_mode.u_3405_b_manual_request;
IF _w18 THEN u_3405_b_speed_request := opc.popa_0092_u_3405_b_hmi_speed_request; END_IF
_w19 := general.ed_routine_maint AND maint_mode.u_3405_b_maint_request;
IF _w19 THEN u_3405_b_speed_request := opc.popa_0092_u_3405_b_hmi_speed_request; END_IF
_w20 := (((_w17 OR u_3405_b_enable AND general.ed_routine_stop) AND NOT gen_alm_active OR _w18) AND NOT interlocks.u_3405_b_intlk OR _w19) AND NOT stopping_mode.u_3405_b_stop_request;
u_3405_b_enable := _w20;
u_3405_b_ons(CLK := _w20); // R_TRIG
u_3405_b_pid_reset := u_3405_b_ons.Q;

// NETWORK 23
u_3405_b(
    run_feedback := io_mapping.u_3405_b_run_feedback,
    runtime_maint_reset := opc.popa_0092_u_3405_b_runtime_maint_reset,
    run_request := pump_manager.u_3405_b_enable,
    speed_request := u_3405_b_speed_request,
    speed_feedback := io_mapping.u_3405_b_speed_feedback.scaled_value,
    fault := faults.u_3405_b_fail_to_start.active OR faults.u_3405_b_fail_to_stop.active,
    daily_reset := general.daily_reset); // motor_vfd

// NETWORK 24
opc.popa_0092_u_3405_b_runtime_maint_Reset R= opc.popa_0092_u_3405_b_runtime_maint_Reset;

// NETWORK 25 (disabled)
// label: Pump u_3160 - enable, and output logic

// NETWORK 26
IF NOT u_3160_b_enable THEN opc.popa_0082_u_3160_b_hmi_speed_request := 0; END_IF

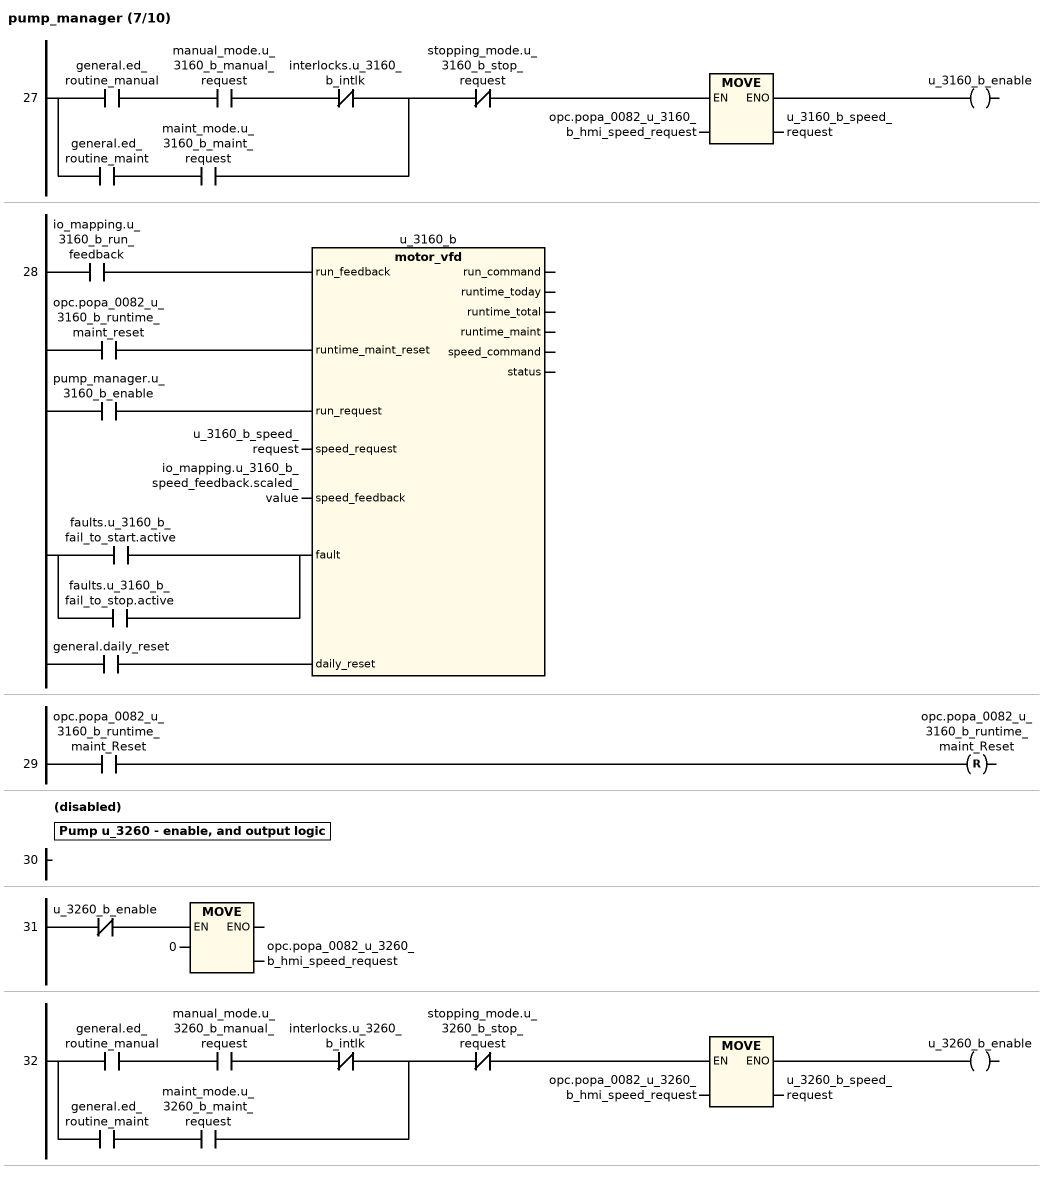
// NETWORK 27
_w21 := (general.ed_routine_manual AND manual_mode.u_3160_b_manual_request AND NOT interlocks.u_3160_b_intlk OR general.ed_routine_maint AND maint_mode.u_3160_b_maint_request) AND NOT stopping_mode.u_3160_b_stop_request;
IF _w21 THEN u_3160_b_speed_request := opc.popa_0082_u_3160_b_hmi_speed_request; END_IF
u_3160_b_enable := _w21;

// NETWORK 28
u_3160_b(
    run_feedback := io_mapping.u_3160_b_run_feedback,
    runtime_maint_reset := opc.popa_0082_u_3160_b_runtime_maint_reset,
    run_request := pump_manager.u_3160_b_enable,
    speed_request := u_3160_b_speed_request,
    speed_feedback := io_mapping.u_3160_b_speed_feedback.scaled_value,
    fault := faults.u_3160_b_fail_to_start.active OR faults.u_3160_b_fail_to_stop.active,
    daily_reset := general.daily_reset); // motor_vfd

// NETWORK 29
opc.popa_0082_u_3160_b_runtime_maint_Reset R= opc.popa_0082_u_3160_b_runtime_maint_Reset;

// NETWORK 30 (disabled)
// label: Pump u_3260 - enable, and output logic

// NETWORK 31
IF NOT u_3260_b_enable THEN opc.popa_0082_u_3260_b_hmi_speed_request := 0; END_IF

// NETWORK 32
_w22 := (general.ed_routine_manual AND manual_mode.u_3260_b_manual_request AND NOT interlocks.u_3260_b_intlk OR general.ed_routine_maint AND maint_mode.u_3260_b_maint_request) AND NOT stopping_mode.u_3260_b_stop_request;
IF _w22 THEN u_3260_b_speed_request := opc.popa_0082_u_3260_b_hmi_speed_request; END_IF
u_3260_b_enable := _w22;

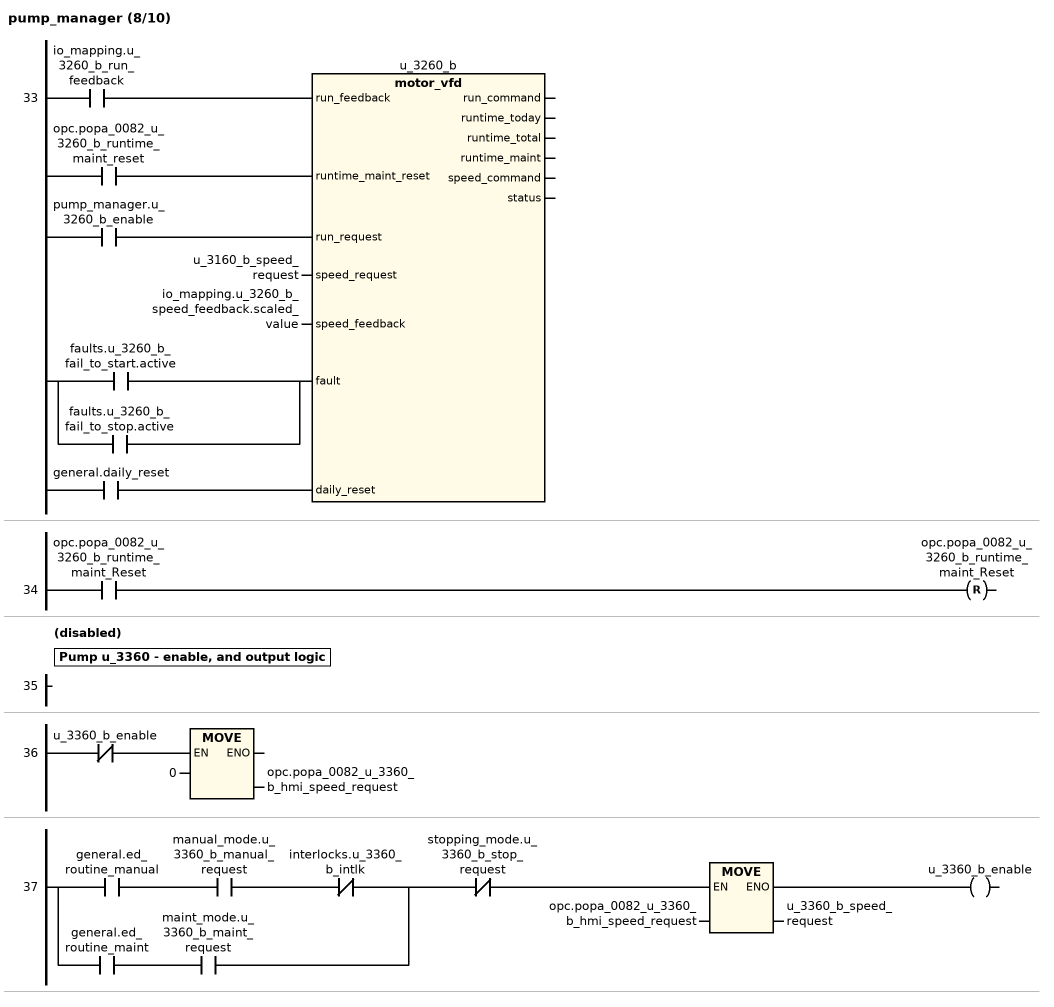
// NETWORK 33
u_3260_b(
    run_feedback := io_mapping.u_3260_b_run_feedback,
    runtime_maint_reset := opc.popa_0082_u_3260_b_runtime_maint_reset,
    run_request := pump_manager.u_3260_b_enable,
    speed_request := u_3160_b_speed_request,
    speed_feedback := io_mapping.u_3260_b_speed_feedback.scaled_value,
    fault := faults.u_3260_b_fail_to_start.active OR faults.u_3260_b_fail_to_stop.active,
    daily_reset := general.daily_reset); // motor_vfd

// NETWORK 34
opc.popa_0082_u_3260_b_runtime_maint_Reset R= opc.popa_0082_u_3260_b_runtime_maint_Reset;

// NETWORK 35 (disabled)
// label: Pump u_3360 - enable, and output logic

// NETWORK 36
IF NOT u_3360_b_enable THEN opc.popa_0082_u_3360_b_hmi_speed_request := 0; END_IF

// NETWORK 37
_w23 := (general.ed_routine_manual AND manual_mode.u_3360_b_manual_request AND NOT interlocks.u_3360_b_intlk OR general.ed_routine_maint AND maint_mode.u_3360_b_maint_request) AND NOT stopping_mode.u_3360_b_stop_request;
IF _w23 THEN u_3360_b_speed_request := opc.popa_0082_u_3360_b_hmi_speed_request; END_IF
u_3360_b_enable := _w23;

